RoboDK station: kr30 cnc 072119 adjusting.rdk

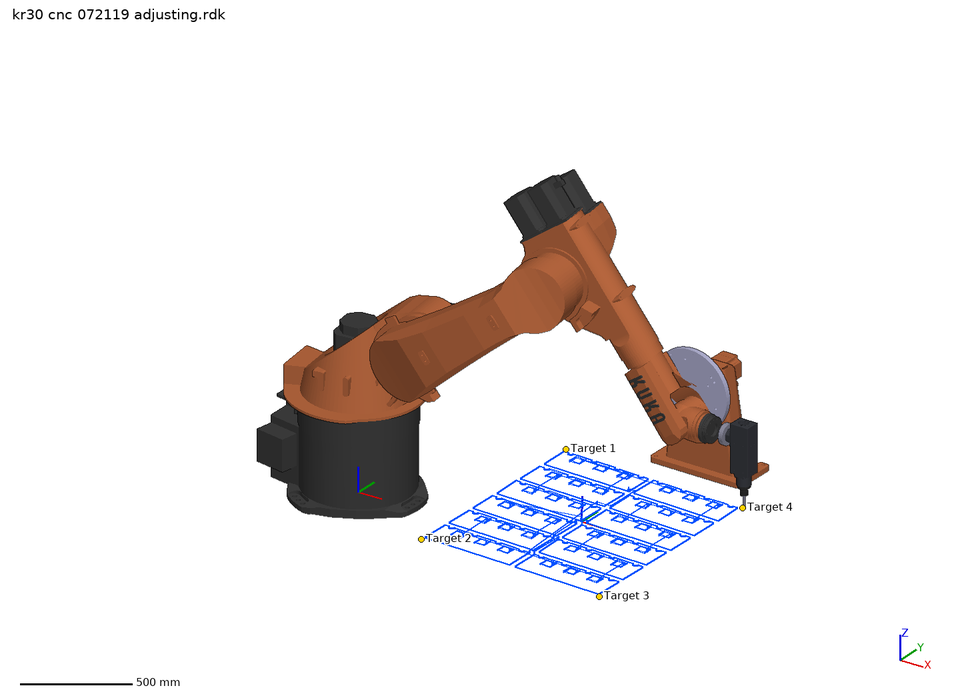
[picture v0: the station drawn from its stored meshes, robots at their saved joint values, targets as dots, program paths as lines]
Station kr30 cnc 072119 adjusting. Poses are relative to the parent item; angles as X-Y-Z fixed-axis rotations.
  - frame GIGASHEEN 7th Axis Base at (0, 0, 0) mm
    - robot KUKA KP1 MD250: 1 axes, payload 250 kg
        modified DH rows (alpha deg, a mm, theta deg, d mm): 0, 0, 0, 0
        base shift (1587.22, 296.05, 828) mm, rotated rx 0 ry 90 rz -90 deg
        joint limits [-3600] to [3600]; home [0]; saved at [1119.52]
      - frame Turntable Base at (243.9, -362.78, 658.66) mm, rotated rx -90.25 ry 0 rz 49.48 deg
  - frame GIGASHEEN Base at (0, 0, 0) mm
    - robot GIGASHEEN (model KUKA KR 30 HA): 6 axes, payload 30 kg, reach 2033 mm, repeatability 0.05 mm, weight 665 kg
        modified DH rows (alpha deg, a mm, theta deg, d mm): 0, 0, 0, 815; -90, 350, 0, 0; 0, 850, -90, 0; -90, 145, 0, 820; 90, 0, 0, 0; -90, 0, 180, 170
        joint limits [-185, -135, -120, -350, -119, -350] to [185, 35, 158, 350, 119, 350]; home [0, -90, 90, 0, 0, 0]; saved at [-6.898, -35.989, 90.741, -8.88, -55.221, 5.167]
      - tool 1/2" End Mill TCP, TCP at (337.71, -2.2, 160.57) mm, rotated rx 0 ry 90 rz 0 deg, size 415.8 x 102 x 153.6 mm
    - target Target 1 (joint target) at (982.46, 202.21, 406.25) mm, rotated rx -179.95 ry 0.15 rz -89.48 deg; joints [7.49, -59.642, 144.935, 97.969, -90.801, -4.608] of GIGASHEEN
    - target Target 2 (joint target) at (986.83, -921.64, 412.07) mm, rotated rx -179.94 ry 0.15 rz -89.48 deg; joints [51.766, -38.608, 94.384, 136.851, -116.554, -22.567] of GIGASHEEN
    - target Target 3 (joint target) at (1949.02, -919.97, 396.91) mm, rotated rx -179.94 ry 0.14 rz 179.61 deg; joints [29.5, -22.76, 62.288, 41.088, -47.759, -30.404] of GIGASHEEN
    - target Target 4 (joint target) at (1949.02, 190.94, 391.63) mm, rotated rx -179.94 ry 0.14 rz 179.61 deg; joints [-6.898, -35.989, 90.741, -8.88, -55.221, 5.167] of GIGASHEEN
  - machining project Machining Settings: C:/Users/liqui/OneDrive/Desktop/first half pipe jig.apt | rotZ(0) | rotX(0)*rotY(0) | rotZ(0)
  - program Machining (1954 instructions, listed below)
  - program Prog2 (4 instructions, listed below)
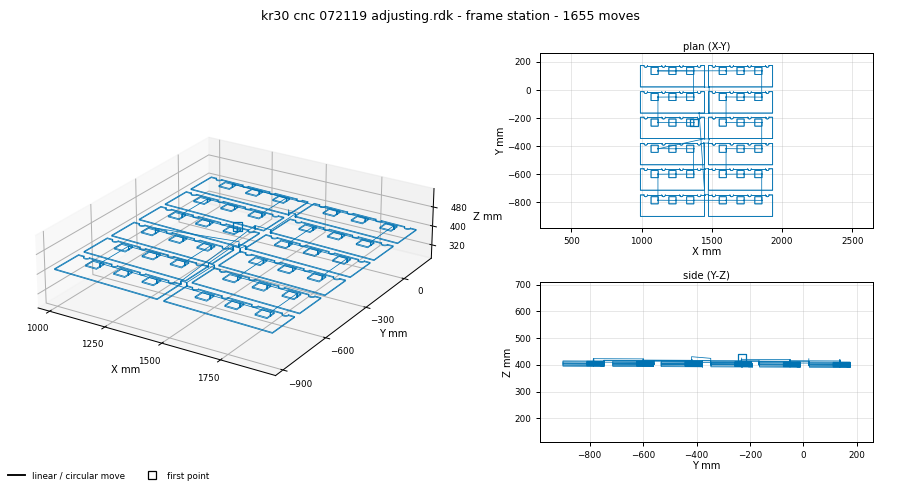
[picture p0: tool path of kr30 cnc 072119 adjusting.rdk in frame station, 1655 of 1659 moves have a stored position in this frame; points joined in program order, loops and branches not executed]

--- program Machining (robot GIGASHEEN) ---
  Smooth(0)
  Set Ref.: Turntable Base
  Set Tool: 1/2" End Mill TCP
  Show 1/2" End Mill TCP
  Print: /'1001'
  Print: /''
  Print: /'2D Contour2'
  Set speed (500.0 mm/s)
  MoveJ 1 to (-92.16, 131.49, 15) mm, rotated rx -180 ry 0 rz -179 deg; joints [17.436, -76.67, 121.961, 23.843, -47.841, -16.522]
  MoveL 2 to (-92.16, 131.49, 15) mm, rotated rx -180 ry 0 rz -179 deg; joints [17.436, -76.67, 121.961, 23.843, -47.841, -16.522]
  MoveL 3 to (-92.16, 131.49, 15) mm, rotated rx -180 ry 0 rz -179 deg; joints [17.436, -76.67, 121.961, 23.843, -47.841, -16.522]
  Set speed (500.0 mm/s)
  MoveL 4 to (-92.16, 131.49, 6) mm, rotated rx 180 ry 0 rz -179 deg; joints [17.436, -76.289, 122.229, 23.608, -48.436, -16.171]
  Set speed (25.4 mm/s)
  MoveL 5 to (-92.16, 131.49, -3.54) mm, rotated rx 180 ry 0 rz -179 deg; joints [17.436, -75.878, 122.507, 23.368, -49.068, -15.806]
  MoveC 6 to (-91.98, 131.48, -3.99) mm, rotated rx -180 ry 0 rz -179 deg; joints [17.434, -75.848, 122.506, 23.355, -49.094, -15.788] to (-91.53, 131.49, -4.17) mm, rotated rx -180 ry 0 rz -179 deg; joints [17.428, -75.815, 122.478, 23.345, -49.097, -15.78]
  Set speed (50.8 mm/s)
  MoveL 7 to (-90.89, 131.49, -4.18) mm, rotated rx -180 ry 0 rz -179 deg; joints [17.42, -75.779, 122.432, 23.338, -49.085, -15.779]
  MoveC 8 to (-90.44, 131.3, -4.18) mm, rotated rx -180 ry 0 rz -179 deg; joints [17.422, -75.751, 122.395, 23.344, -49.077, -15.786] to (-90.26, 130.85, -4.17) mm, rotated rx -180 ry 0 rz -179 deg; joints [17.44, -75.733, 122.371, 23.369, -49.077, -15.803]
  MoveL 9 to (-90.26, 105.45, -4.18) mm, rotated rx 180 ry 0 rz -179 deg; joints [18.57, -75.299, 121.799, 24.851, -49.269, -16.815]
  MoveL 10 to (-141.06, 105.45, -4.17) mm, rotated rx -180 ry 0 rz -179 deg; joints [19.31, -78.143, 125.477, 25.479, -50.238, -16.95]
  MoveL 11 to (-141.06, 156.25, -4.17) mm, rotated rx -180 ry 0 rz -179 deg; joints [16.952, -79.034, 126.595, 22.442, -49.797, -14.928]
  MoveL 12 to (-90.26, 156.25, -4.17) mm, rotated rx -180 ry 0 rz -179 deg; joints [16.296, -76.14, 122.904, 21.865, -48.892, -14.78]
  MoveL 13 to (-90.26, 130.85, -4.17) mm, rotated rx -180 ry 0 rz -179 deg; joints [17.44, -75.733, 122.371, 23.369, -49.077, -15.803]
  MoveC 14 to (-90.44, 130.4, -4.17) mm, rotated rx -180 ry 0 rz -179 deg; joints [17.462, -75.736, 122.375, 23.397, -49.084, -15.822] to (-90.89, 130.21, -4.18) mm, rotated rx -180 ry 0 rz -179 deg; joints [17.477, -75.758, 122.404, 23.413, -49.094, -15.83]
  MoveL 15 to (-91.53, 130.21, -4.18) mm, rotated rx 180 ry 0 rz -179 deg; joints [17.485, -75.794, 122.451, 23.42, -49.107, -15.831]
  MoveC 16 to (-91.98, 130.22, -3.99) mm, rotated rx -180 ry 0 rz -179 deg; joints [17.491, -75.827, 122.479, 23.429, -49.103, -15.839] to (-92.16, 130.22, -3.54) mm, rotated rx -180 ry 0 rz -179 deg; joints [17.493, -75.857, 122.479, 23.442, -49.077, -15.857]
  Set speed (500.0 mm/s)
  MoveL 17 to (-92.16, 130.22, 5) mm, rotated rx -180 ry 0 rz -179 deg; joints [17.493, -76.225, 122.231, 23.658, -48.512, -16.184]
  MoveL 18 to (-92.16, 131.49, 5) mm, rotated rx 180 ry 0 rz -179 deg; joints [17.436, -76.246, 122.259, 23.583, -48.502, -16.132]
  Set speed (25.4 mm/s)
  MoveL 19 to (-92.16, 131.49, 1.82) mm, rotated rx -180 ry 0 rz -179 deg; joints [17.436, -76.11, 122.352, 23.502, -48.712, -16.01]
  MoveL 20 to (-92.16, 131.49, -7.72) mm, rotated rx -180 ry 0 rz -179 deg; joints [17.436, -75.696, 122.626, 23.265, -49.345, -15.648]
  MoveC 21 to (-91.98, 131.49, -8.16) mm, rotated rx 180 ry 0 rz -179 deg; joints [17.434, -75.666, 122.625, 23.252, -49.371, -15.631] to (-91.53, 131.49, -8.35) mm, rotated rx -180 ry 0 rz -179 deg; joints [17.428, -75.632, 122.597, 23.242, -49.374, -15.623]
  Set speed (50.8 mm/s)
  MoveL 22 to (-90.89, 131.49, -8.35) mm, rotated rx -180 ry 0 rz -179 deg; joints [17.42, -75.597, 122.551, 23.235, -49.362, -15.622]
  MoveC 23 to (-90.44, 131.3, -8.35) mm, rotated rx -180 ry 0 rz -179 deg; joints [17.422, -75.569, 122.513, 23.242, -49.354, -15.629] to (-90.26, 130.85, -8.35) mm, rotated rx 180 ry 0 rz -179 deg; joints [17.44, -75.551, 122.49, 23.266, -49.354, -15.646]
  MoveL 24 to (-90.26, 105.45, -8.35) mm, rotated rx -180 ry 0 rz -179 deg; joints [18.57, -75.118, 121.917, 24.743, -49.54, -16.65]
  MoveL 25 to (-141.06, 105.45, -8.35) mm, rotated rx -180 ry 0 rz -179 deg; joints [19.31, -77.953, 125.598, 25.368, -50.519, -16.777]
  MoveL 26 to (-141.06, 156.25, -8.35) mm, rotated rx -180 ry 0 rz -179 deg; joints [16.952, -78.842, 126.718, 22.341, -50.089, -14.771]
  MoveL 27 to (-90.26, 156.25, -8.35) mm, rotated rx 180 ry 0 rz -179 deg; joints [16.296, -75.956, 123.023, 21.767, -49.173, -14.631]
  MoveL 28 to (-90.26, 130.85, -8.35) mm, rotated rx 180 ry 0 rz -179 deg; joints [17.44, -75.551, 122.49, 23.266, -49.354, -15.646]
  MoveC 29 to (-90.44, 130.4, -8.35) mm, rotated rx -180 ry 0 rz -179 deg; joints [17.462, -75.554, 122.494, 23.294, -49.36, -15.664] to (-90.89, 130.21, -8.35) mm, rotated rx -180 ry 0 rz -179 deg; joints [17.477, -75.576, 122.523, 23.31, -49.371, -15.672]
  MoveL 30 to (-91.53, 130.21, -8.35) mm, rotated rx -180 ry 0 rz -179 deg; joints [17.485, -75.611, 122.57, 23.317, -49.383, -15.673]
  MoveC 31 to (-91.98, 130.22, -8.16) mm, rotated rx 180 ry 0 rz -179 deg; joints [17.491, -75.645, 122.598, 23.326, -49.38, -15.681] to (-92.16, 130.22, -7.72) mm, rotated rx -180 ry 0 rz -179 deg; joints [17.493, -75.675, 122.598, 23.339, -49.354, -15.698]
  Set speed (500.0 mm/s)
  MoveL 32 to (-92.16, 130.22, 6) mm, rotated rx 180 ry 0 rz -179 deg; joints [17.493, -76.268, 122.202, 23.684, -48.446, -16.223]
  MoveL 33 to (-219.16, 131.49, 6) mm, rotated rx -180 ry 0 rz -179 deg; joints [19.301, -83.624, 131.192, 25.384, -50.447, -16.812]
  Set speed (25.4 mm/s)
  MoveL 34 to (-219.16, 131.49, -3.54) mm, rotated rx -180 ry 0 rz -179 deg; joints [19.301, -83.162, 131.493, 25.118, -51.137, -16.392]
  MoveC 35 to (-218.98, 131.49, -3.99) mm, rotated rx -180 ry 0 rz -179 deg; joints [19.298, -83.129, 131.494, 25.103, -51.167, -16.371] to (-218.53, 131.48, -4.17) mm, rotated rx -180 ry 0 rz -179 deg; joints [19.29, -83.093, 131.469, 25.09, -51.175, -16.359]
  Set speed (50.8 mm/s)
  MoveL 36 to (-217.89, 131.49, -4.18) mm, rotated rx -180 ry 0 rz -179 deg; joints [19.28, -83.056, 131.426, 25.079, -51.167, -16.355]
  MoveC 37 to (-217.44, 131.3, -4.17) mm, rotated rx -180 ry 0 rz -179 deg; joints [19.282, -83.026, 131.392, 25.083, -51.163, -16.359] to (-217.26, 130.85, -4.17) mm, rotated rx -180 ry 0 rz -179 deg; joints [19.301, -83.006, 131.369, 25.108, -51.166, -16.375]
  MoveL 38 to (-217.26, 105.45, -4.17) mm, rotated rx -180 ry 0 rz -179 deg; joints [20.54, -82.498, 130.777, 26.656, -51.45, -17.372]
  MoveL 39 to (-268.06, 105.45, -4.18) mm, rotated rx 180 ry 0 rz -179 deg; joints [21.453, -85.484, 134.171, 27.617, -52.089, -17.82]
  MoveL 40 to (-268.06, 156.25, -4.18) mm, rotated rx 180 ry 0 rz -179 deg; joints [18.856, -86.551, 135.335, 24.418, -51.424, -15.806]
  MoveL 41 to (-217.26, 156.25, -4.18) mm, rotated rx -180 ry 0 rz -179 deg; joints [18.043, -83.485, 131.921, 23.527, -50.889, -15.358]
  MoveL 42 to (-217.26, 130.85, -4.17) mm, rotated rx -180 ry 0 rz -179 deg; joints [19.301, -83.006, 131.369, 25.108, -51.166, -16.375]
  MoveC 43 to (-217.44, 130.4, -4.18) mm, rotated rx 180 ry 0 rz -179 deg; joints [19.326, -83.008, 131.371, 25.138, -51.173, -16.394] to (-217.89, 130.22, -4.17) mm, rotated rx -180 ry 0 rz -179 deg; joints [19.342, -83.031, 131.398, 25.157, -51.181, -16.405]
  MoveL 44 to (-218.53, 130.22, -4.18) mm, rotated rx 180 ry 0 rz -179 deg; joints [19.353, -83.068, 131.441, 25.168, -51.189, -16.41]
  MoveC 45 to (-218.98, 130.21, -3.99) mm, rotated rx -180 ry 0 rz -179 deg; joints [19.36, -83.104, 131.466, 25.181, -51.182, -16.421] to (-219.16, 130.21, -3.54) mm, rotated rx -180 ry 0 rz -179 deg; joints [19.363, -83.137, 131.464, 25.196, -51.151, -16.442]
  Set speed (500.0 mm/s)
  MoveL 46 to (-219.16, 130.22, 5) mm, rotated rx 180 ry 0 rz -179 deg; joints [19.363, -83.551, 131.196, 25.434, -50.534, -16.819]
  MoveL 47 to (-219.16, 131.48, 5) mm, rotated rx -180 ry 0 rz -179 deg; joints [19.301, -83.576, 131.224, 25.355, -50.519, -16.768]
  Set speed (25.4 mm/s)
  MoveL 48 to (-219.16, 131.48, 1.82) mm, rotated rx -180 ry 0 rz -179 deg; joints [19.301, -83.423, 131.325, 25.266, -50.749, -16.627]
  MoveL 49 to (-219.16, 131.49, -7.72) mm, rotated rx -180 ry 0 rz -179 deg; joints [19.301, -82.956, 131.622, 25.004, -51.44, -16.21]
  MoveC 50 to (-218.98, 131.49, -8.16) mm, rotated rx -180 ry 0 rz -179 deg; joints [19.298, -82.923, 131.623, 24.989, -51.47, -16.189] to (-218.53, 131.49, -8.35) mm, rotated rx -180 ry 0 rz -179 deg; joints [19.29, -82.888, 131.598, 24.977, -51.478, -16.178]
  Set speed (50.8 mm/s)
  MoveL 51 to (-217.89, 131.48, -8.35) mm, rotated rx -180 ry 0 rz -179 deg; joints [19.28, -82.85, 131.555, 24.966, -51.47, -16.174]
  MoveC 52 to (-217.44, 131.3, -8.35) mm, rotated rx -180 ry 0 rz -179 deg; joints [19.282, -82.82, 131.52, 24.97, -51.466, -16.178] to (-217.26, 130.85, -8.35) mm, rotated rx -180 ry 0 rz -179 deg; joints [19.301, -82.801, 131.497, 24.994, -51.468, -16.194]
  MoveL 53 to (-217.26, 105.45, -8.35) mm, rotated rx -180 ry 0 rz -179 deg; joints [20.54, -82.294, 130.905, 26.539, -51.747, -17.182]
  MoveL 54 to (-268.06, 105.45, -8.35) mm, rotated rx -180 ry 0 rz -179 deg; joints [21.453, -85.271, 134.303, 27.493, -52.396, -17.618]
  MoveL 55 to (-268.06, 156.25, -8.35) mm, rotated rx -180 ry 0 rz -179 deg; joints [18.856, -86.334, 135.469, 24.303, -51.745, -15.621]
  MoveL 56 to (-217.26, 156.25, -8.35) mm, rotated rx -180 ry 0 rz -179 deg; joints [18.043, -83.278, 132.05, 23.419, -51.197, -15.185]
  MoveL 57 to (-217.26, 130.85, -8.35) mm, rotated rx -180 ry 0 rz -179 deg; joints [19.301, -82.801, 131.497, 24.994, -51.468, -16.194]
  MoveC 58 to (-217.44, 130.4, -8.35) mm, rotated rx -180 ry 0 rz -179 deg; joints [19.326, -82.803, 131.5, 25.025, -51.476, -16.213] to (-217.89, 130.22, -8.35) mm, rotated rx 180 ry 0 rz -179 deg; joints [19.342, -82.826, 131.526, 25.044, -51.484, -16.223]
  MoveL 59 to (-218.53, 130.21, -8.35) mm, rotated rx -180 ry 0 rz -179 deg; joints [19.353, -82.863, 131.57, 25.055, -51.492, -16.228]
  MoveC 60 to (-218.98, 130.21, -8.16) mm, rotated rx -180 ry 0 rz -179 deg; joints [19.36, -82.898, 131.595, 25.067, -51.484, -16.239] to (-219.16, 130.22, -7.72) mm, rotated rx 180 ry 0 rz -179 deg; joints [19.363, -82.932, 131.593, 25.082, -51.454, -16.26]
  Set speed (500.0 mm/s)
  MoveL 61 to (-219.16, 130.21, 6) mm, rotated rx -180 ry 0 rz -179 deg; joints [19.363, -83.599, 131.164, 25.462, -50.462, -16.863]
  MoveL 62 to (-346.16, 131.48, 6) mm, rotated rx -180 ry 0 rz -179 deg; joints [21.621, -91.451, 139.452, 28.072, -51.536, -18.353]
  Set speed (25.4 mm/s)
  MoveL 63 to (-346.16, 131.48, -3.54) mm, rotated rx -180 ry 0 rz -179 deg; joints [21.621, -90.932, 139.786, 27.76, -52.288, -17.847]
  MoveC 64 to (-345.98, 131.49, -3.99) mm, rotated rx 180 ry 0 rz -179 deg; joints [21.617, -90.896, 139.79, 27.741, -52.323, -17.82] to (-345.53, 131.48, -4.17) mm, rotated rx -180 ry 0 rz -179 deg; joints [21.608, -90.857, 139.768, 27.724, -52.335, -17.803]
  Set speed (50.8 mm/s)
  MoveL 65 to (-344.89, 131.49, -4.18) mm, rotated rx -180 ry 0 rz -179 deg; joints [21.595, -90.816, 139.728, 27.708, -52.332, -17.793]
  MoveC 66 to (-344.44, 131.3, -4.17) mm, rotated rx 180 ry 0 rz -179 deg; joints [21.596, -90.783, 139.696, 27.709, -52.333, -17.793] to (-344.26, 130.85, -4.18) mm, rotated rx 180 ry 0 rz -179 deg; joints [21.617, -90.76, 139.673, 27.733, -52.339, -17.808]
  MoveL 67 to (-344.26, 105.45, -4.17) mm, rotated rx -180 ry 0 rz -179 deg; joints [22.984, -90.134, 139.054, 29.366, -52.775, -18.799]
  MoveL 68 to (-395.06, 105.45, -4.18) mm, rotated rx -180 ry 0 rz -179 deg; joints [24.132, -93.379, 142.168, 30.774, -53.04, -19.7]
  MoveL 69 to (-395.06, 156.25, -4.18) mm, rotated rx -180 ry 0 rz -179 deg; joints [21.254, -94.725, 143.389, 27.385, -52.009, -17.686]
  MoveL 70 to (-344.26, 156.25, -4.18) mm, rotated rx -180 ry 0 rz -179 deg; joints [20.224, -91.353, 140.251, 26.054, -51.913, -16.782]
  MoveL 71 to (-344.26, 130.85, -4.18) mm, rotated rx 180 ry 0 rz -179 deg; joints [21.617, -90.76, 139.673, 27.733, -52.339, -17.808]
  MoveC 72 to (-344.44, 130.4, -4.18) mm, rotated rx -180 ry 0 rz -179 deg; joints [21.645, -90.761, 139.674, 27.767, -52.348, -17.829] to (-344.89, 130.22, -4.18) mm, rotated rx -180 ry 0 rz -179 deg; joints [21.664, -90.786, 139.698, 27.79, -52.354, -17.843]
  MoveL 73 to (-345.53, 130.22, -4.18) mm, rotated rx 180 ry 0 rz -179 deg; joints [21.677, -90.826, 139.738, 27.806, -52.357, -17.853]
  MoveC 74 to (-345.98, 130.21, -3.99) mm, rotated rx 180 ry 0 rz -179 deg; joints [21.686, -90.865, 139.76, 27.824, -52.344, -17.87] to (-346.16, 130.22, -3.54) mm, rotated rx -180 ry 0 rz -179 deg; joints [21.69, -90.902, 139.756, 27.843, -52.31, -17.897]
  Set speed (500.0 mm/s)
  MoveL 75 to (-346.16, 130.22, 5) mm, rotated rx -180 ry 0 rz -179 deg; joints [21.69, -91.366, 139.458, 28.123, -51.637, -18.351]
  MoveL 76 to (-346.16, 131.48, 5) mm, rotated rx -180 ry 0 rz -179 deg; joints [21.621, -91.397, 139.488, 28.039, -51.614, -18.3]
  Set speed (25.4 mm/s)
  MoveL 77 to (-346.16, 131.49, 1.83) mm, rotated rx -180 ry 0 rz -179 deg; joints [21.621, -91.225, 139.599, 27.934, -51.864, -18.13]
  MoveL 78 to (-346.16, 131.49, -7.72) mm, rotated rx 180 ry 0 rz -179 deg; joints [21.621, -90.702, 139.929, 27.626, -52.619, -17.627]
  MoveC 79 to (-345.98, 131.49, -8.16) mm, rotated rx 180 ry 0 rz -179 deg; joints [21.617, -90.665, 139.933, 27.607, -52.654, -17.601] to (-345.53, 131.49, -8.35) mm, rotated rx 180 ry 0 rz -179 deg; joints [21.608, -90.626, 139.911, 27.59, -52.666, -17.584]
  Set speed (50.8 mm/s)
  MoveL 80 to (-344.89, 131.48, -8.35) mm, rotated rx -180 ry 0 rz -179 deg; joints [21.595, -90.585, 139.871, 27.575, -52.663, -17.575]
  MoveC 81 to (-344.44, 131.3, -8.35) mm, rotated rx -180 ry 0 rz -179 deg; joints [21.596, -90.552, 139.838, 27.576, -52.664, -17.575] to (-344.26, 130.85, -8.35) mm, rotated rx 180 ry 0 rz -179 deg; joints [21.617, -90.53, 139.816, 27.6, -52.67, -17.59]
  MoveL 82 to (-344.26, 105.45, -8.35) mm, rotated rx -180 ry 0 rz -179 deg; joints [22.984, -89.906, 139.195, 29.229, -53.097, -18.572]
  MoveL 83 to (-395.06, 105.45, -8.35) mm, rotated rx 180 ry 0 rz -179 deg; joints [24.132, -93.14, 142.316, 30.626, -53.373, -19.453]
  MoveL 84 to (-395.06, 156.25, -8.35) mm, rotated rx -180 ry 0 rz -179 deg; joints [21.254, -94.482, 143.541, 27.245, -52.359, -17.457]
  MoveL 85 to (-344.26, 156.25, -8.35) mm, rotated rx -180 ry 0 rz -179 deg; joints [20.224, -91.12, 140.395, 25.925, -52.251, -16.573]
  MoveL 86 to (-344.26, 130.85, -8.35) mm, rotated rx 180 ry 0 rz -179 deg; joints [21.617, -90.53, 139.816, 27.6, -52.67, -17.59]
  MoveC 87 to (-344.44, 130.4, -8.35) mm, rotated rx -180 ry 0 rz -179 deg; joints [21.645, -90.531, 139.817, 27.634, -52.679, -17.61] to (-344.89, 130.21, -8.35) mm, rotated rx 180 ry 0 rz -179 deg; joints [21.664, -90.555, 139.841, 27.657, -52.684, -17.624]
  MoveL 88 to (-345.53, 130.22, -8.35) mm, rotated rx -180 ry 0 rz -179 deg; joints [21.677, -90.595, 139.881, 27.673, -52.688, -17.634]
  MoveC 89 to (-345.98, 130.22, -8.16) mm, rotated rx 180 ry 0 rz -179 deg; joints [21.686, -90.634, 139.903, 27.69, -52.675, -17.651] to (-346.16, 130.21, -7.72) mm, rotated rx -180 ry 0 rz -179 deg; joints [21.69, -90.671, 139.899, 27.709, -52.641, -17.677]
  Set speed (500.0 mm/s)
  MoveL 90 to (-346.16, 130.22, 6) mm, rotated rx 180 ry 0 rz -179 deg; joints [21.69, -91.42, 139.423, 28.156, -51.558, -18.405]
  MoveL 91 to (-346.16, 313.35, 6) mm, rotated rx -180 ry 0 rz -179 deg; joints [11.148, -94.869, 142.627, 14.906, -48.733, -9.958]
  Set speed (25.4 mm/s)
  MoveL 92 to (-346.16, 313.36, -3.54) mm, rotated rx 180 ry 0 rz -179 deg; joints [11.148, -94.327, 142.977, 14.709, -49.594, -9.657]
  MoveC 93 to (-345.98, 313.36, -3.99) mm, rotated rx 180 ry 0 rz -179 deg; joints [11.146, -94.288, 142.981, 14.697, -49.636, -9.641] to (-345.53, 313.35, -4.17) mm, rotated rx -180 ry 0 rz -179 deg; joints [11.142, -94.246, 142.959, 14.687, -49.655, -9.63]
  Set speed (50.8 mm/s)
  MoveL 94 to (-344.89, 313.36, -4.18) mm, rotated rx 180 ry 0 rz -179 deg; joints [11.135, -94.201, 142.919, 14.677, -49.658, -9.623]
  MoveC 95 to (-344.44, 313.17, -4.18) mm, rotated rx -180 ry 0 rz -179 deg; joints [11.141, -94.167, 142.888, 14.684, -49.662, -9.627] to (-344.26, 312.72, -4.18) mm, rotated rx -180 ry 0 rz -179 deg; joints [11.166, -94.148, 142.871, 14.716, -49.668, -9.648]
  MoveL 96 to (-344.26, 287.32, -4.18) mm, rotated rx 180 ry 0 rz -179 deg; joints [12.685, -93.803, 142.558, 16.665, -49.969, -10.899]
  MoveL 97 to (-395.06, 287.32, -4.18) mm, rotated rx -180 ry 0 rz -179 deg; joints [13.345, -97.456, 145.743, 17.629, -49.652, -11.626]
  MoveL 98 to (-395.06, 338.12, -4.18) mm, rotated rx -180 ry 0 rz -179 deg; joints [10.127, -98.178, 146.337, 13.482, -48.954, -8.947]
  MoveL 99 to (-344.26, 338.12, -4.17) mm, rotated rx -180 ry 0 rz -179 deg; joints [9.633, -94.446, 143.14, 12.732, -49.4, -8.365]
  MoveL 100 to (-344.26, 312.72, -4.17) mm, rotated rx -180 ry 0 rz -179 deg; joints [11.166, -94.148, 142.871, 14.716, -49.668, -9.648]
  MoveC 101 to (-344.44, 312.27, -4.18) mm, rotated rx -180 ry 0 rz -179 deg; joints [11.195, -94.155, 142.878, 14.754, -49.672, -9.672] to (-344.89, 312.09, -4.18) mm, rotated rx 180 ry 0 rz -179 deg; joints [11.211, -94.185, 142.904, 14.775, -49.672, -9.686]
  MoveL 102 to (-345.53, 312.09, -4.18) mm, rotated rx -180 ry 0 rz -179 deg; joints [11.218, -94.23, 142.945, 14.785, -49.669, -9.694]
  MoveC 103 to (-345.98, 312.09, -3.99) mm, rotated rx -180 ry 0 rz -179 deg; joints [11.223, -94.272, 142.967, 14.796, -49.65, -9.705] to (-346.16, 312.08, -3.54) mm, rotated rx -180 ry 0 rz -179 deg; joints [11.225, -94.311, 142.962, 14.808, -49.609, -9.721]
  Set speed (500.0 mm/s)
  MoveL 104 to (-346.16, 312.09, 5) mm, rotated rx 180 ry 0 rz -179 deg; joints [11.225, -94.796, 142.65, 14.985, -48.838, -9.992]
  MoveL 105 to (-346.16, 313.36, 5) mm, rotated rx 180 ry 0 rz -179 deg; joints [11.148, -94.813, 142.664, 14.885, -48.823, -9.926]
  Set speed (25.4 mm/s)
  MoveL 106 to (-346.16, 313.36, 1.82) mm, rotated rx -180 ry 0 rz -179 deg; joints [11.148, -94.633, 142.781, 14.819, -49.109, -9.826]
  MoveL 107 to (-346.16, 313.35, -7.71) mm, rotated rx -180 ry 0 rz -179 deg; joints [11.148, -94.086, 143.128, 14.625, -49.974, -9.527]
  MoveC 108 to (-345.98, 313.36, -8.16) mm, rotated rx -180 ry 0 rz -179 deg; joints [11.146, -94.047, 143.132, 14.614, -50.015, -9.511] to (-345.53, 313.36, -8.35) mm, rotated rx -180 ry 0 rz -179 deg; joints [11.142, -94.004, 143.11, 14.603, -50.034, -9.501]
  Set speed (50.8 mm/s)
  MoveL 109 to (-344.89, 313.35, -8.35) mm, rotated rx -180 ry 0 rz -179 deg; joints [11.135, -93.959, 143.069, 14.593, -50.037, -9.494]
  MoveC 110 to (-344.44, 313.17, -8.35) mm, rotated rx -180 ry 0 rz -179 deg; joints [11.141, -93.925, 143.038, 14.601, -50.041, -9.498] to (-344.26, 312.72, -8.35) mm, rotated rx -180 ry 0 rz -179 deg; joints [11.166, -93.907, 143.021, 14.633, -50.047, -9.518]
  MoveL 111 to (-344.26, 287.32, -8.35) mm, rotated rx -180 ry 0 rz -179 deg; joints [12.685, -93.563, 142.707, 16.572, -50.342, -10.754]
  MoveL 112 to (-395.06, 287.32, -8.35) mm, rotated rx -180 ry 0 rz -179 deg; joints [13.345, -97.205, 145.9, 17.525, -50.041, -11.464]
  MoveL 113 to (-395.06, 338.12, -8.35) mm, rotated rx 180 ry 0 rz -179 deg; joints [10.127, -97.925, 146.497, 13.399, -49.355, -8.82]
  MoveL 114 to (-344.26, 338.12, -8.35) mm, rotated rx -180 ry 0 rz -179 deg; joints [9.633, -94.204, 143.291, 12.658, -49.783, -8.251]
  MoveL 115 to (-344.26, 312.72, -8.35) mm, rotated rx -180 ry 0 rz -179 deg; joints [11.166, -93.907, 143.021, 14.633, -50.047, -9.518]
  MoveC 116 to (-344.44, 312.27, -8.35) mm, rotated rx -180 ry 0 rz -179 deg; joints [11.195, -93.914, 143.028, 14.67, -50.051, -9.542] to (-344.89, 312.08, -8.35) mm, rotated rx -180 ry 0 rz -179 deg; joints [11.211, -93.943, 143.054, 14.691, -50.051, -9.556]
  MoveL 117 to (-345.53, 312.08, -8.35) mm, rotated rx -180 ry 0 rz -179 deg; joints [11.218, -93.988, 143.095, 14.701, -50.048, -9.563]
  MoveC 118 to (-345.98, 312.08, -8.16) mm, rotated rx -180 ry 0 rz -179 deg; joints [11.223, -94.031, 143.117, 14.712, -50.029, -9.574] to (-346.16, 312.08, -7.72) mm, rotated rx -180 ry 0 rz -179 deg; joints [11.225, -94.07, 143.113, 14.724, -49.988, -9.59]
  Set speed (500.0 mm/s)
  MoveL 119 to (-346.16, 312.08, 6) mm, rotated rx -180 ry 0 rz -179 deg; joints [11.225, -94.852, 142.613, 15.006, -48.748, -10.024]
  MoveL 120 to (-219.16, 313.36, 6) mm, rotated rx -180 ry 0 rz -179 deg; joints [9.941, -86.348, 134.223, 13.295, -48.648, -8.873]
  Set speed (25.4 mm/s)
  MoveL 121 to (-219.16, 313.36, -3.54) mm, rotated rx -180 ry 0 rz -179 deg; joints [9.941, -85.865, 134.534, 13.138, -49.421, -8.633]
  MoveC 122 to (-218.98, 313.36, -3.99) mm, rotated rx 180 ry 0 rz -179 deg; joints [9.939, -85.831, 134.535, 13.129, -49.456, -8.621] to (-218.53, 313.36, -4.17) mm, rotated rx -180 ry 0 rz -179 deg; joints [9.935, -85.793, 134.51, 13.121, -49.468, -8.614]
  Set speed (50.8 mm/s)
  MoveL 123 to (-217.89, 313.36, -4.17) mm, rotated rx -180 ry 0 rz -179 deg; joints [9.93, -85.753, 134.466, 13.115, -49.463, -8.611]
  MoveC 124 to (-217.44, 313.17, -4.18) mm, rotated rx 180 ry 0 rz -179 deg; joints [9.936, -85.723, 134.433, 13.124, -49.461, -8.617] to (-217.26, 312.72, -4.18) mm, rotated rx 180 ry 0 rz -179 deg; joints [9.959, -85.707, 134.416, 13.153, -49.463, -8.636]
  MoveL 125 to (-217.26, 287.32, -4.17) mm, rotated rx -180 ry 0 rz -179 deg; joints [11.305, -85.436, 134.118, 14.905, -49.652, -9.777]
  MoveL 126 to (-268.06, 287.32, -4.18) mm, rotated rx 180 ry 0 rz -179 deg; joints [11.816, -88.674, 137.573, 15.516, -49.95, -10.128]
  MoveL 127 to (-268.06, 338.12, -4.18) mm, rotated rx 180 ry 0 rz -179 deg; joints [8.984, -89.225, 138.138, 11.846, -49.523, -7.754]
  MoveL 128 to (-217.26, 338.12, -4.18) mm, rotated rx -180 ry 0 rz -179 deg; joints [8.602, -85.94, 134.672, 11.38, -49.294, -7.478]
  MoveL 129 to (-217.26, 312.72, -4.18) mm, rotated rx 180 ry 0 rz -179 deg; joints [9.959, -85.707, 134.416, 13.153, -49.463, -8.636]
  MoveC 130 to (-217.44, 312.27, -4.17) mm, rotated rx -180 ry 0 rz -179 deg; joints [9.984, -85.714, 134.424, 13.186, -49.467, -8.657] to (-217.89, 312.08, -4.17) mm, rotated rx -180 ry 0 rz -179 deg; joints [9.998, -85.74, 134.453, 13.203, -49.472, -8.668]
  MoveL 131 to (-218.53, 312.08, -4.18) mm, rotated rx -180 ry 0 rz -179 deg; joints [10.003, -85.78, 134.497, 13.209, -49.477, -8.671]
  MoveC 132 to (-218.98, 312.08, -3.99) mm, rotated rx -180 ry 0 rz -179 deg; joints [10.007, -85.818, 134.522, 13.217, -49.465, -8.679] to (-219.16, 312.08, -3.54) mm, rotated rx 180 ry 0 rz -179 deg; joints [10.008, -85.853, 134.52, 13.226, -49.43, -8.691]
  Set speed (500.0 mm/s)
  MoveL 133 to (-219.16, 312.08, 5) mm, rotated rx -180 ry 0 rz -179 deg; joints [10.008, -86.285, 134.242, 13.368, -48.739, -8.907]
  MoveL 134 to (-219.16, 313.35, 5) mm, rotated rx -180 ry 0 rz -179 deg; joints [9.941, -86.298, 134.256, 13.278, -48.729, -8.848]
  Set speed (25.4 mm/s)
  MoveL 135 to (-219.16, 313.36, 1.82) mm, rotated rx -180 ry 0 rz -179 deg; joints [9.941, -86.138, 134.36, 13.226, -48.986, -8.768]
  MoveL 136 to (-219.16, 313.35, -7.72) mm, rotated rx -180 ry 0 rz -179 deg; joints [9.941, -85.651, 134.668, 13.07, -49.759, -8.53]
  MoveC 137 to (-218.98, 313.36, -8.16) mm, rotated rx -180 ry 0 rz -179 deg; joints [9.939, -85.616, 134.669, 13.062, -49.794, -8.517] to (-218.53, 313.36, -8.35) mm, rotated rx -180 ry 0 rz -179 deg; joints [9.935, -85.579, 134.644, 13.054, -49.806, -8.511]
  Set speed (50.8 mm/s)
  MoveL 138 to (-217.89, 313.36, -8.35) mm, rotated rx 180 ry 0 rz -179 deg; joints [9.93, -85.539, 134.6, 13.048, -49.802, -8.507]
  MoveC 139 to (-217.44, 313.17, -8.35) mm, rotated rx 180 ry 0 rz -179 deg; joints [9.936, -85.509, 134.567, 13.057, -49.799, -8.513] to (-217.26, 312.72, -8.35) mm, rotated rx -180 ry 0 rz -179 deg; joints [9.959, -85.493, 134.549, 13.086, -49.801, -8.533]
  MoveL 140 to (-217.26, 287.32, -8.35) mm, rotated rx -180 ry 0 rz -179 deg; joints [11.305, -85.223, 134.251, 14.83, -49.986, -9.661]
  MoveL 141 to (-268.06, 287.32, -8.35) mm, rotated rx 180 ry 0 rz -179 deg; joints [11.816, -88.45, 137.712, 15.435, -50.3, -10.002]
  MoveL 142 to (-268.06, 338.12, -8.35) mm, rotated rx -180 ry 0 rz -179 deg; joints [8.984, -88.999, 138.277, 11.783, -49.88, -7.656]
  MoveL 143 to (-217.26, 338.12, -8.35) mm, rotated rx -180 ry 0 rz -179 deg; joints [8.602, -85.725, 134.805, 11.321, -49.636, -7.388]
  MoveL 144 to (-217.26, 312.72, -8.35) mm, rotated rx -180 ry 0 rz -179 deg; joints [9.959, -85.493, 134.549, 13.086, -49.801, -8.533]
  MoveC 145 to (-217.44, 312.27, -8.35) mm, rotated rx -180 ry 0 rz -179 deg; joints [9.984, -85.5, 134.557, 13.119, -49.806, -8.554] to (-217.89, 312.08, -8.35) mm, rotated rx 180 ry 0 rz -179 deg; joints [9.998, -85.526, 134.586, 13.136, -49.81, -8.564]
  MoveL 146 to (-218.53, 312.09, -8.35) mm, rotated rx -180 ry 0 rz -179 deg; joints [10.003, -85.566, 134.63, 13.142, -49.815, -8.567]
  MoveC 147 to (-218.98, 312.08, -8.16) mm, rotated rx -180 ry 0 rz -179 deg; joints [10.007, -85.604, 134.655, 13.149, -49.803, -8.574] to (-219.16, 312.08, -7.72) mm, rotated rx -180 ry 0 rz -179 deg; joints [10.008, -85.639, 134.654, 13.158, -49.768, -8.587]
  Set speed (500.0 mm/s)
  MoveL 148 to (-219.16, 312.08, 6) mm, rotated rx -180 ry 0 rz -179 deg; joints [10.008, -86.335, 134.209, 13.384, -48.658, -8.932]
  MoveL 149 to (-92.16, 313.35, 6) mm, rotated rx -180 ry 0 rz -179 deg; joints [8.988, -78.58, 125.15, 12.287, -47.233, -8.413]
  Set speed (25.4 mm/s)
  MoveL 150 to (-92.16, 313.36, -3.54) mm, rotated rx 180 ry 0 rz -179 deg; joints [8.988, -78.153, 125.434, 12.15, -47.928, -8.209]
  MoveC 151 to (-91.98, 313.36, -3.99) mm, rotated rx -180 ry 0 rz -179 deg; joints [8.987, -78.121, 125.433, 12.142, -47.957, -8.199] to (-91.53, 313.36, -4.17) mm, rotated rx -180 ry 0 rz -179 deg; joints [8.984, -78.087, 125.405, 12.137, -47.964, -8.194]
  Set speed (50.8 mm/s)
  MoveL 152 to (-90.89, 313.36, -4.18) mm, rotated rx 180 ry 0 rz -179 deg; joints [8.98, -78.049, 125.358, 12.133, -47.953, -8.193]
  MoveC 153 to (-90.44, 313.17, -4.17) mm, rotated rx -180 ry 0 rz -179 deg; joints [8.986, -78.021, 125.323, 12.142, -47.947, -8.201] to (-90.26, 312.72, -4.17) mm, rotated rx -180 ry 0 rz -179 deg; joints [9.006, -78.007, 125.304, 12.17, -47.946, -8.22]
  MoveL 154 to (-90.26, 287.32, -4.17) mm, rotated rx 180 ry 0 rz -179 deg; joints [10.214, -77.781, 125.018, 13.789, -48.071, -9.313]
  MoveL 155 to (-141.06, 287.32, -4.17) mm, rotated rx -180 ry 0 rz -179 deg; joints [10.621, -80.783, 128.739, 14.172, -48.835, -9.437]
  MoveL 156 to (-141.06, 338.12, -4.17) mm, rotated rx -180 ry 0 rz -179 deg; joints [8.094, -81.231, 129.278, 10.825, -48.558, -7.213]
  MoveL 157 to (-90.26, 338.12, -4.17) mm, rotated rx -180 ry 0 rz -179 deg; joints [7.791, -78.201, 125.55, 10.538, -47.834, -7.118]
  MoveL 158 to (-90.26, 312.72, -4.17) mm, rotated rx -180 ry 0 rz -179 deg; joints [9.006, -78.007, 125.304, 12.17, -47.946, -8.22]
  MoveC 159 to (-90.44, 312.27, -4.17) mm, rotated rx -180 ry 0 rz -179 deg; joints [9.028, -78.014, 125.314, 12.2, -47.951, -8.24] to (-90.89, 312.09, -4.17) mm, rotated rx -180 ry 0 rz -179 deg; joints [9.04, -78.039, 125.345, 12.215, -47.959, -8.248]
  MoveL 160 to (-91.53, 312.09, -4.18) mm, rotated rx 180 ry 0 rz -179 deg; joints [9.045, -78.076, 125.392, 12.218, -47.97, -8.249]
  MoveC 161 to (-91.98, 312.09, -3.99) mm, rotated rx 180 ry 0 rz -179 deg; joints [9.048, -78.111, 125.42, 12.224, -47.963, -8.254] to (-92.16, 312.09, -3.54) mm, rotated rx -180 ry 0 rz -179 deg; joints [9.049, -78.142, 125.421, 12.231, -47.934, -8.264]
  Set speed (500.0 mm/s)
  MoveL 162 to (-92.16, 312.09, 5) mm, rotated rx -180 ry 0 rz -179 deg; joints [9.049, -78.525, 125.167, 12.355, -47.312, -8.447]
  MoveL 163 to (-92.16, 313.36, 5) mm, rotated rx 180 ry 0 rz -179 deg; joints [8.988, -78.535, 125.18, 12.273, -47.306, -8.391]
  Set speed (25.4 mm/s)
  MoveL 164 to (-92.16, 313.36, 1.82) mm, rotated rx -180 ry 0 rz -179 deg; joints [8.988, -78.394, 125.275, 12.227, -47.537, -8.323]
  MoveL 165 to (-92.16, 313.36, -7.71) mm, rotated rx 180 ry 0 rz -179 deg; joints [8.988, -77.963, 125.556, 12.091, -48.232, -8.121]
  MoveC 166 to (-91.98, 313.36, -8.16) mm, rotated rx -180 ry 0 rz -179 deg; joints [8.987, -77.932, 125.555, 12.084, -48.262, -8.111] to (-91.53, 313.36, -8.35) mm, rotated rx -180 ry 0 rz -179 deg; joints [8.984, -77.897, 125.527, 12.079, -48.268, -8.107]
  Set speed (50.8 mm/s)
  MoveL 167 to (-90.89, 313.36, -8.35) mm, rotated rx 180 ry 0 rz -179 deg; joints [8.98, -77.86, 125.48, 12.075, -48.258, -8.106]
  MoveC 168 to (-90.44, 313.17, -8.35) mm, rotated rx -180 ry 0 rz -179 deg; joints [8.986, -77.832, 125.445, 12.084, -48.251, -8.113] to (-90.26, 312.72, -8.35) mm, rotated rx -180 ry 0 rz -179 deg; joints [9.006, -77.817, 125.426, 12.111, -48.25, -8.132]
  MoveL 169 to (-90.26, 287.32, -8.35) mm, rotated rx -180 ry 0 rz -179 deg; joints [10.214, -77.593, 125.14, 13.723, -48.372, -9.214]
  MoveL 170 to (-141.06, 287.32, -8.35) mm, rotated rx -180 ry 0 rz -179 deg; joints [10.621, -80.585, 128.864, 14.104, -49.149, -9.333]
  MoveL 171 to (-141.06, 338.12, -8.35) mm, rotated rx -180 ry 0 rz -179 deg; joints [8.094, -81.032, 129.404, 10.772, -48.877, -7.132]
  MoveL 172 to (-90.26, 338.12, -8.35) mm, rotated rx 180 ry 0 rz -179 deg; joints [7.791, -78.011, 125.672, 10.486, -48.141, -7.041]
  MoveL 173 to (-90.26, 312.72, -8.35) mm, rotated rx -180 ry 0 rz -179 deg; joints [9.006, -77.817, 125.426, 12.111, -48.25, -8.132]
  MoveC 174 to (-90.44, 312.27, -8.35) mm, rotated rx 180 ry 0 rz -179 deg; joints [9.028, -77.825, 125.435, 12.141, -48.255, -8.152] to (-90.89, 312.09, -8.35) mm, rotated rx 180 ry 0 rz -179 deg; joints [9.04, -77.849, 125.467, 12.156, -48.263, -8.16]
  MoveL 175 to (-91.53, 312.08, -8.35) mm, rotated rx -180 ry 0 rz -179 deg; joints [9.045, -77.887, 125.514, 12.159, -48.274, -8.161]
  MoveC 176 to (-91.98, 312.09, -8.16) mm, rotated rx -180 ry 0 rz -179 deg; joints [9.048, -77.921, 125.542, 12.165, -48.268, -8.166] to (-92.16, 312.08, -7.72) mm, rotated rx -180 ry 0 rz -179 deg; joints [9.049, -77.953, 125.543, 12.172, -48.238, -8.175]
  Set speed (500.0 mm/s)
  MoveL 177 to (-92.16, 312.09, 6) mm, rotated rx -180 ry 0 rz -179 deg; joints [9.049, -78.569, 125.137, 12.37, -47.239, -8.469]
  MoveL 178 to (-92.16, 499.69, 6) mm, rotated rx -180 ry 0 rz -179 deg; joints [-0.04, -79.259, 125.995, -0.054, -46.737, 0.037]
  Set speed (25.4 mm/s)
  MoveL 179 to (-92.16, 499.69, -3.54) mm, rotated rx 180 ry 0 rz -179 deg; joints [-0.04, -78.827, 126.281, -0.054, -47.454, 0.036]
  MoveC 180 to (-91.98, 499.69, -3.99) mm, rotated rx -180 ry 0 rz -179 deg; joints [-0.039, -78.795, 126.281, -0.054, -47.485, 0.036] to (-91.53, 499.69, -4.17) mm, rotated rx -180 ry 0 rz -179 deg; joints [-0.039, -78.76, 126.253, -0.053, -47.493, 0.036]
  Set speed (50.8 mm/s)
  MoveL 181 to (-90.89, 499.69, -4.18) mm, rotated rx -180 ry 0 rz -179 deg; joints [-0.039, -78.722, 126.205, -0.052, -47.483, 0.035]
  MoveC 182 to (-90.44, 499.51, -4.17) mm, rotated rx -180 ry 0 rz -179 deg; joints [-0.029, -78.696, 126.172, -0.039, -47.476, 0.027] to (-90.26, 499.06, -4.17) mm, rotated rx 180 ry 0 rz -179 deg; joints [-0.007, -78.685, 126.159, -0.01, -47.474, 0.006]
  MoveL 183 to (-90.26, 473.66, -4.18) mm, rotated rx 180 ry 0 rz -179 deg; joints [1.229, -78.695, 126.172, 1.667, -47.488, -1.126]
  MoveL 184 to (-141.06, 473.66, -4.17) mm, rotated rx -180 ry 0 rz -179 deg; joints [1.239, -81.761, 129.909, 1.663, -48.16, -1.109]
  MoveL 185 to (-141.06, 524.46, -4.18) mm, rotated rx 180 ry 0 rz -179 deg; joints [-1.343, -81.704, 129.842, -1.803, -48.152, 1.203]
  MoveL 186 to (-90.26, 524.46, -4.18) mm, rotated rx -180 ry 0 rz -179 deg; joints [-1.242, -78.642, 126.105, -1.685, -47.475, 1.139]
  MoveL 187 to (-90.26, 499.06, -4.17) mm, rotated rx 180 ry 0 rz -179 deg; joints [-0.007, -78.685, 126.159, -0.01, -47.474, 0.006]
  MoveC 188 to (-90.44, 498.61, -4.17) mm, rotated rx 180 ry 0 rz -179 deg; joints [0.015, -78.697, 126.173, 0.02, -47.477, -0.013] to (-90.89, 498.42, -4.18) mm, rotated rx -180 ry 0 rz -179 deg; joints [0.023, -78.724, 126.207, 0.032, -47.483, -0.021]
  MoveL 189 to (-91.53, 498.42, -4.17) mm, rotated rx 180 ry 0 rz -179 deg; joints [0.023, -78.761, 126.254, 0.031, -47.493, -0.021]
  MoveC 190 to (-91.98, 498.42, -3.99) mm, rotated rx -180 ry 0 rz -179 deg; joints [0.022, -78.797, 126.282, 0.03, -47.486, -0.021] to (-92.16, 498.42, -3.54) mm, rotated rx 180 ry 0 rz -179 deg; joints [0.022, -78.828, 126.283, 0.03, -47.455, -0.02]
  Set speed (500.0 mm/s)
  MoveL 191 to (-92.16, 498.42, 5) mm, rotated rx -180 ry 0 rz -179 deg; joints [0.022, -79.215, 126.027, 0.031, -46.812, -0.021]
  MoveL 192 to (-92.16, 499.69, 5) mm, rotated rx -180 ry 0 rz -179 deg; joints [-0.04, -79.214, 126.026, -0.054, -46.812, 0.037]
  Set speed (25.4 mm/s)
  MoveL 193 to (-92.16, 499.69, 1.83) mm, rotated rx 180 ry 0 rz -179 deg; joints [-0.04, -79.071, 126.121, -0.054, -47.051, 0.037]
  MoveL 194 to (-92.16, 499.69, -7.72) mm, rotated rx -180 ry 0 rz -179 deg; joints [-0.04, -78.636, 126.404, -0.054, -47.769, 0.036]
  MoveC 195 to (-91.98, 499.69, -8.16) mm, rotated rx -180 ry 0 rz -179 deg; joints [-0.039, -78.604, 126.403, -0.053, -47.8, 0.036] to (-91.53, 499.69, -8.35) mm, rotated rx 180 ry 0 rz -179 deg; joints [-0.039, -78.569, 126.375, -0.053, -47.807, 0.035]
  Set speed (50.8 mm/s)
  MoveL 196 to (-90.89, 499.69, -8.35) mm, rotated rx 180 ry 0 rz -179 deg; joints [-0.039, -78.531, 126.328, -0.052, -47.797, 0.035]
  MoveC 197 to (-90.44, 499.51, -8.35) mm, rotated rx 180 ry 0 rz -179 deg; joints [-0.029, -78.504, 126.295, -0.039, -47.79, 0.026] to (-90.26, 499.06, -8.35) mm, rotated rx -180 ry 0 rz -179 deg; joints [-0.007, -78.494, 126.281, -0.01, -47.787, 0.006]
  MoveL 198 to (-90.26, 473.66, -8.35) mm, rotated rx -180 ry 0 rz -179 deg; joints [1.229, -78.504, 126.294, 1.658, -47.802, -1.114]
  MoveL 199 to (-141.06, 473.66, -8.35) mm, rotated rx -180 ry 0 rz -179 deg; joints [1.239, -81.56, 130.036, 1.655, -48.488, -1.097]
  MoveL 200 to (-141.06, 524.46, -8.35) mm, rotated rx -180 ry 0 rz -179 deg; joints [-1.343, -81.503, 129.968, -1.793, -48.479, 1.189]
  MoveL 201 to (-90.26, 524.46, -8.35) mm, rotated rx -180 ry 0 rz -179 deg; joints [-1.242, -78.451, 126.227, -1.677, -47.789, 1.127]
  MoveL 202 to (-90.26, 499.06, -8.35) mm, rotated rx -180 ry 0 rz -179 deg; joints [-0.007, -78.494, 126.281, -0.01, -47.787, 0.006]
  MoveC 203 to (-90.44, 498.61, -8.35) mm, rotated rx -180 ry 0 rz -179 deg; joints [0.015, -78.505, 126.296, 0.02, -47.79, -0.013] to (-90.89, 498.42, -8.35) mm, rotated rx 180 ry 0 rz -179 deg; joints [0.023, -78.532, 126.329, 0.031, -47.797, -0.021]
  MoveL 204 to (-91.53, 498.42, -8.35) mm, rotated rx 180 ry 0 rz -179 deg; joints [0.023, -78.57, 126.377, 0.031, -47.807, -0.021]
  MoveC 205 to (-91.98, 498.42, -8.16) mm, rotated rx -180 ry 0 rz -179 deg; joints [0.022, -78.605, 126.405, 0.03, -47.8, -0.02] to (-92.16, 498.42, -7.72) mm, rotated rx -180 ry 0 rz -179 deg; joints [0.022, -78.637, 126.406, 0.03, -47.769, -0.02]
  Set speed (500.0 mm/s)
  MoveL 206 to (-92.16, 498.42, 6) mm, rotated rx -180 ry 0 rz -179 deg; joints [0.022, -79.26, 125.997, 0.031, -46.737, -0.021]
  MoveL 207 to (-219.16, 499.69, 6) mm, rotated rx -180 ry 0 rz -179 deg; joints [-0.165, -87.168, 135.103, -0.223, -47.935, 0.149]
  Set speed (25.4 mm/s)
  MoveL 208 to (-219.16, 499.69, -3.54) mm, rotated rx 180 ry 0 rz -179 deg; joints [-0.165, -86.68, 135.417, -0.22, -48.738, 0.145]
  MoveC 209 to (-218.98, 499.69, -3.99) mm, rotated rx -180 ry 0 rz -179 deg; joints [-0.165, -86.645, 135.419, -0.22, -48.775, 0.145] to (-218.53, 499.69, -4.17) mm, rotated rx -180 ry 0 rz -179 deg; joints [-0.165, -86.606, 135.394, -0.219, -48.788, 0.144]
  Set speed (50.8 mm/s)
  MoveL 210 to (-217.89, 499.69, -4.18) mm, rotated rx -180 ry 0 rz -179 deg; joints [-0.164, -86.565, 135.35, -0.218, -48.785, 0.144]
  MoveC 211 to (-217.44, 499.51, -4.18) mm, rotated rx -180 ry 0 rz -179 deg; joints [-0.153, -86.536, 135.319, -0.204, -48.783, 0.134] to (-217.26, 499.06, -4.18) mm, rotated rx -180 ry 0 rz -179 deg; joints [-0.129, -86.525, 135.307, -0.171, -48.782, 0.113]
  MoveL 212 to (-217.26, 473.66, -4.18) mm, rotated rx -180 ry 0 rz -179 deg; joints [1.256, -86.537, 135.32, 1.67, -48.795, -1.1]
  MoveL 213 to (-268.06, 473.66, -4.18) mm, rotated rx -180 ry 0 rz -179 deg; joints [1.269, -89.88, 138.799, 1.684, -48.932, -1.106]
  MoveL 214 to (-268.06, 524.46, -4.17) mm, rotated rx -180 ry 0 rz -179 deg; joints [-1.64, -89.809, 138.728, -2.175, -48.94, 1.429]
  MoveL 215 to (-217.26, 524.46, -4.17) mm, rotated rx -180 ry 0 rz -179 deg; joints [-1.512, -86.473, 135.25, -2.01, -48.795, 1.325]
  MoveL 216 to (-217.26, 499.06, -4.18) mm, rotated rx -180 ry 0 rz -179 deg; joints [-0.129, -86.525, 135.307, -0.171, -48.782, 0.113]
  MoveC 217 to (-217.44, 498.61, -4.18) mm, rotated rx 180 ry 0 rz -179 deg; joints [-0.104, -86.538, 135.32, -0.139, -48.783, 0.092] to (-217.89, 498.42, -4.17) mm, rotated rx -180 ry 0 rz -179 deg; joints [-0.095, -86.567, 135.352, -0.126, -48.785, 0.083]
  MoveL 218 to (-218.53, 498.42, -4.18) mm, rotated rx -180 ry 0 rz -179 deg; joints [-0.095, -86.608, 135.396, -0.127, -48.788, 0.084]
  MoveC 219 to (-218.98, 498.42, -3.99) mm, rotated rx 180 ry 0 rz -179 deg; joints [-0.096, -86.646, 135.421, -0.128, -48.775, 0.084] to (-219.16, 498.42, -3.54) mm, rotated rx -180 ry 0 rz -179 deg; joints [-0.096, -86.681, 135.419, -0.128, -48.738, 0.084]
  Set speed (500.0 mm/s)
  MoveL 220 to (-219.16, 498.42, 5) mm, rotated rx 180 ry 0 rz -179 deg; joints [-0.096, -87.119, 135.138, -0.129, -48.019, 0.086]
  MoveL 221 to (-219.16, 499.69, 5) mm, rotated rx -180 ry 0 rz -179 deg; joints [-0.165, -87.117, 135.136, -0.223, -48.019, 0.149]
  Set speed (25.4 mm/s)
  MoveL 222 to (-219.16, 499.69, 1.82) mm, rotated rx -180 ry 0 rz -179 deg; joints [-0.165, -86.956, 135.241, -0.222, -48.286, 0.148]
  MoveL 223 to (-219.16, 499.69, -7.72) mm, rotated rx -180 ry 0 rz -179 deg; joints [-0.165, -86.463, 135.552, -0.219, -49.09, 0.143]
  MoveC 224 to (-218.98, 499.69, -8.16) mm, rotated rx -180 ry 0 rz -179 deg; joints [-0.165, -86.427, 135.554, -0.219, -49.127, 0.143] to (-218.53, 499.69, -8.35) mm, rotated rx -180 ry 0 rz -179 deg; joints [-0.165, -86.389, 135.529, -0.218, -49.14, 0.143]
  Set speed (50.8 mm/s)
  MoveL 225 to (-217.89, 499.69, -8.35) mm, rotated rx 180 ry 0 rz -179 deg; joints [-0.164, -86.348, 135.485, -0.217, -49.137, 0.142]
  MoveC 226 to (-217.44, 499.51, -8.35) mm, rotated rx 180 ry 0 rz -179 deg; joints [-0.153, -86.32, 135.454, -0.203, -49.134, 0.133] to (-217.26, 499.06, -8.35) mm, rotated rx -180 ry 0 rz -179 deg; joints [-0.129, -86.308, 135.441, -0.17, -49.133, 0.111]
  MoveL 227 to (-217.26, 473.66, -8.35) mm, rotated rx 180 ry 0 rz -179 deg; joints [1.256, -86.321, 135.455, 1.661, -49.146, -1.087]
  MoveL 228 to (-268.06, 473.66, -8.35) mm, rotated rx 180 ry 0 rz -179 deg; joints [1.269, -89.652, 138.94, 1.674, -49.3, -1.092]
  MoveL 229 to (-268.06, 524.46, -8.35) mm, rotated rx -180 ry 0 rz -179 deg; joints [-1.64, -89.581, 138.869, -2.163, -49.308, 1.411]
  MoveL 230 to (-217.26, 524.46, -8.35) mm, rotated rx 180 ry 0 rz -179 deg; joints [-1.512, -86.256, 135.385, -2, -49.146, 1.308]
  MoveL 231 to (-217.26, 499.06, -8.35) mm, rotated rx -180 ry 0 rz -179 deg; joints [-0.129, -86.308, 135.441, -0.17, -49.133, 0.111]
  MoveC 232 to (-217.44, 498.61, -8.35) mm, rotated rx -180 ry 0 rz -179 deg; joints [-0.104, -86.321, 135.455, -0.138, -49.134, 0.09] to (-217.89, 498.42, -8.35) mm, rotated rx -180 ry 0 rz -179 deg; joints [-0.095, -86.35, 135.486, -0.125, -49.137, 0.082]
  MoveL 233 to (-218.53, 498.42, -8.35) mm, rotated rx -180 ry 0 rz -179 deg; joints [-0.095, -86.391, 135.53, -0.126, -49.14, 0.083]
  MoveC 234 to (-218.98, 498.42, -8.16) mm, rotated rx -180 ry 0 rz -179 deg; joints [-0.096, -86.429, 135.556, -0.127, -49.127, 0.083] to (-219.16, 498.42, -7.72) mm, rotated rx -180 ry 0 rz -179 deg; joints [-0.096, -86.464, 135.554, -0.127, -49.09, 0.083]
  Set speed (500.0 mm/s)
  MoveL 235 to (-219.16, 498.42, 6) mm, rotated rx -180 ry 0 rz -179 deg; joints [-0.096, -87.169, 135.105, -0.129, -47.935, 0.087]
  MoveL 236 to (-346.16, 499.69, 6) mm, rotated rx -180 ry 0 rz -179 deg; joints [-0.326, -95.921, 143.551, -0.441, -47.632, 0.297]
  Set speed (25.4 mm/s)
  MoveL 237 to (-346.16, 499.69, -3.54) mm, rotated rx -180 ry 0 rz -179 deg; joints [-0.326, -95.372, 143.907, -0.435, -48.535, 0.288]
  MoveC 238 to (-345.98, 499.69, -3.99) mm, rotated rx -180 ry 0 rz -179 deg; joints [-0.326, -95.333, 143.911, -0.434, -48.58, 0.287] to (-345.53, 499.69, -4.17) mm, rotated rx 180 ry 0 rz -179 deg; joints [-0.325, -95.289, 143.889, -0.433, -48.601, 0.287]
  Set speed (50.8 mm/s)
  MoveL 239 to (-344.89, 499.69, -4.17) mm, rotated rx -180 ry 0 rz -179 deg; joints [-0.324, -95.243, 143.848, -0.432, -48.607, 0.286]
  MoveC 240 to (-344.44, 499.51, -4.17) mm, rotated rx 180 ry 0 rz -179 deg; joints [-0.312, -95.21, 143.82, -0.416, -48.611, 0.275] to (-344.26, 499.06, -4.18) mm, rotated rx -180 ry 0 rz -179 deg; joints [-0.284, -95.197, 143.809, -0.378, -48.612, 0.25]
  MoveL 241 to (-344.26, 473.66, -4.17) mm, rotated rx -180 ry 0 rz -179 deg; joints [1.291, -95.213, 143.823, 1.721, -48.622, -1.138]
  MoveL 242 to (-395.06, 473.66, -4.17) mm, rotated rx 180 ry 0 rz -179 deg; joints [1.308, -99.043, 147.034, 1.761, -48.005, -1.178]
  MoveL 243 to (-395.06, 524.46, -4.18) mm, rotated rx -180 ry 0 rz -179 deg; joints [-2.023, -98.949, 146.96, -2.721, -48.043, 1.82]
  MoveL 244 to (-344.26, 524.46, -4.17) mm, rotated rx 180 ry 0 rz -179 deg; joints [-1.857, -95.13, 143.749, -2.475, -48.646, 1.636]
  MoveL 245 to (-344.26, 499.06, -4.18) mm, rotated rx -180 ry 0 rz -179 deg; joints [-0.284, -95.197, 143.809, -0.378, -48.612, 0.25]
  MoveC 246 to (-344.44, 498.61, -4.17) mm, rotated rx 180 ry 0 rz -179 deg; joints [-0.256, -95.212, 143.821, -0.342, -48.61, 0.226] to (-344.89, 498.42, -4.18) mm, rotated rx -180 ry 0 rz -179 deg; joints [-0.245, -95.245, 143.85, -0.327, -48.606, 0.216]
  MoveL 247 to (-345.53, 498.42, -4.17) mm, rotated rx -180 ry 0 rz -179 deg; joints [-0.246, -95.291, 143.891, -0.328, -48.601, 0.217]
  MoveC 248 to (-345.98, 498.42, -3.99) mm, rotated rx 180 ry 0 rz -179 deg; joints [-0.247, -95.335, 143.913, -0.329, -48.579, 0.218] to (-346.16, 498.42, -3.54) mm, rotated rx -180 ry 0 rz -179 deg; joints [-0.247, -95.374, 143.909, -0.33, -48.535, 0.218]
  Set speed (500.0 mm/s)
  MoveL 249 to (-346.16, 498.42, 5) mm, rotated rx 180 ry 0 rz -179 deg; joints [-0.247, -95.866, 143.591, -0.334, -47.725, 0.225]
  MoveL 250 to (-346.16, 499.69, 5) mm, rotated rx -180 ry 0 rz -179 deg; joints [-0.326, -95.864, 143.589, -0.441, -47.726, 0.296]
  Set speed (25.4 mm/s)
  MoveL 251 to (-346.16, 499.69, 1.83) mm, rotated rx -180 ry 0 rz -179 deg; joints [-0.326, -95.682, 143.708, -0.438, -48.026, 0.293]
  MoveL 252 to (-346.16, 499.69, -7.71) mm, rotated rx 180 ry 0 rz -179 deg; joints [-0.326, -95.128, 144.06, -0.432, -48.933, 0.284]
  MoveC 253 to (-345.98, 499.69, -8.16) mm, rotated rx 180 ry 0 rz -179 deg; joints [-0.326, -95.088, 144.064, -0.432, -48.977, 0.283] to (-345.53, 499.69, -8.35) mm, rotated rx 180 ry 0 rz -179 deg; joints [-0.325, -95.044, 144.042, -0.431, -48.998, 0.283]
  Set speed (50.8 mm/s)
  MoveL 254 to (-344.89, 499.69, -8.35) mm, rotated rx -180 ry 0 rz -179 deg; joints [-0.324, -94.998, 144.001, -0.43, -49.004, 0.282]
  MoveC 255 to (-344.44, 499.51, -8.35) mm, rotated rx -180 ry 0 rz -179 deg; joints [-0.312, -94.966, 143.972, -0.413, -49.007, 0.271] to (-344.26, 499.06, -8.35) mm, rotated rx 180 ry 0 rz -179 deg; joints [-0.284, -94.953, 143.961, -0.376, -49.009, 0.247]
  MoveL 256 to (-344.26, 473.66, -8.35) mm, rotated rx 180 ry 0 rz -179 deg; joints [1.291, -94.969, 143.975, 1.711, -49.019, -1.122]
  MoveL 257 to (-395.06, 473.66, -8.35) mm, rotated rx 180 ry 0 rz -179 deg; joints [1.308, -98.787, 147.196, 1.749, -48.422, -1.161]
  MoveL 258 to (-395.06, 524.46, -8.35) mm, rotated rx -180 ry 0 rz -179 deg; joints [-2.023, -98.694, 147.121, -2.704, -48.459, 1.794]
  MoveL 259 to (-344.26, 524.46, -8.35) mm, rotated rx -180 ry 0 rz -179 deg; joints [-1.857, -94.886, 143.902, -2.46, -49.042, 1.613]
  MoveL 260 to (-344.26, 499.06, -8.35) mm, rotated rx 180 ry 0 rz -179 deg; joints [-0.284, -94.953, 143.961, -0.376, -49.009, 0.247]
  MoveC 261 to (-344.44, 498.61, -8.35) mm, rotated rx 180 ry 0 rz -179 deg; joints [-0.256, -94.967, 143.974, -0.34, -49.007, 0.223] to (-344.89, 498.42, -8.35) mm, rotated rx -180 ry 0 rz -179 deg; joints [-0.245, -95, 144.003, -0.325, -49.003, 0.213]
  MoveL 262 to (-345.53, 498.42, -8.35) mm, rotated rx -180 ry 0 rz -179 deg; joints [-0.246, -95.046, 144.044, -0.326, -48.998, 0.214]
  MoveC 263 to (-345.98, 498.42, -8.16) mm, rotated rx -180 ry 0 rz -179 deg; joints [-0.247, -95.09, 144.066, -0.327, -48.976, 0.215] to (-346.16, 498.42, -7.72) mm, rotated rx -180 ry 0 rz -179 deg; joints [-0.247, -95.13, 144.061, -0.328, -48.932, 0.215]
  Set speed (500.0 mm/s)
  MoveL 264 to (-346.16, 498.42, 6) mm, rotated rx -180 ry 0 rz -179 deg; joints [-0.247, -95.923, 143.553, -0.334, -47.631, 0.225]
  MoveL 265 to (139.15, 499.69, 6) mm, rotated rx -180 ry 0 rz -179 deg; joints [0.131, -65.766, 107.508, 0.197, -41.742, -0.147]
  Set speed (25.4 mm/s)
  MoveL 266 to (139.15, 499.69, -3.54) mm, rotated rx -180 ry 0 rz -179 deg; joints [0.131, -65.422, 107.767, 0.195, -42.345, -0.144]
  MoveC 267 to (139.34, 499.69, -3.99) mm, rotated rx -180 ry 0 rz -179 deg; joints [0.131, -65.395, 107.763, 0.195, -42.368, -0.144] to (139.79, 499.69, -4.17) mm, rotated rx -180 ry 0 rz -179 deg; joints [0.132, -65.362, 107.729, 0.195, -42.367, -0.144]
  Set speed (50.8 mm/s)
  MoveL 268 to (140.42, 499.69, -4.17) mm, rotated rx -180 ry 0 rz -179 deg; joints [0.132, -65.326, 107.674, 0.196, -42.348, -0.145]
  MoveC 269 to (140.87, 499.51, -4.17) mm, rotated rx -180 ry 0 rz -179 deg; joints [0.14, -65.3, 107.635, 0.208, -42.335, -0.154] to (141.06, 499.06, -4.17) mm, rotated rx 180 ry 0 rz -179 deg; joints [0.158, -65.29, 107.62, 0.235, -42.33, -0.174]
  MoveL 270 to (141.06, 473.66, -4.18) mm, rotated rx -180 ry 0 rz -179 deg; joints [1.191, -65.298, 107.632, 1.768, -42.348, -1.307]
  MoveL 271 to (90.26, 473.66, -4.17) mm, rotated rx -180 ry 0 rz -179 deg; joints [1.198, -68.212, 111.946, 1.733, -43.747, -1.252]
  MoveL 272 to (90.26, 524.46, -4.18) mm, rotated rx 180 ry 0 rz -179 deg; joints [-0.944, -68.168, 111.882, -1.366, -43.722, 0.987]
  MoveL 273 to (141.06, 524.46, -4.18) mm, rotated rx 180 ry 0 rz -179 deg; joints [-0.874, -65.255, 107.568, -1.298, -42.32, 0.96]
  MoveL 274 to (141.06, 499.06, -4.17) mm, rotated rx 180 ry 0 rz -179 deg; joints [0.158, -65.29, 107.62, 0.235, -42.33, -0.174]
  MoveC 275 to (140.87, 498.61, -4.17) mm, rotated rx -180 ry 0 rz -179 deg; joints [0.176, -65.301, 107.637, 0.262, -42.336, -0.194] to (140.42, 498.42, -4.18) mm, rotated rx 180 ry 0 rz -179 deg; joints [0.184, -65.327, 107.676, 0.273, -42.349, -0.202]
  MoveL 276 to (139.79, 498.42, -4.17) mm, rotated rx 180 ry 0 rz -179 deg; joints [0.183, -65.363, 107.73, 0.272, -42.367, -0.201]
  MoveC 277 to (139.34, 498.42, -3.99) mm, rotated rx 180 ry 0 rz -179 deg; joints [0.183, -65.396, 107.764, 0.272, -42.369, -0.201] to (139.15, 498.42, -3.54) mm, rotated rx 180 ry 0 rz -179 deg; joints [0.183, -65.423, 107.768, 0.272, -42.346, -0.201]
  Set speed (500.0 mm/s)
  MoveL 278 to (139.15, 498.42, 5) mm, rotated rx -180 ry 0 rz -179 deg; joints [0.183, -65.731, 107.537, 0.274, -41.806, -0.205]
  MoveL 279 to (139.15, 499.69, 5) mm, rotated rx -180 ry 0 rz -179 deg; joints [0.131, -65.73, 107.535, 0.197, -41.805, -0.147]
  Set speed (25.4 mm/s)
  MoveL 280 to (139.15, 499.69, 1.82) mm, rotated rx -180 ry 0 rz -179 deg; joints [0.131, -65.616, 107.622, 0.196, -42.006, -0.146]
  MoveL 281 to (139.15, 499.69, -7.72) mm, rotated rx -180 ry 0 rz -179 deg; joints [0.131, -65.269, 107.878, 0.194, -42.609, -0.143]
  MoveC 282 to (139.34, 499.69, -8.16) mm, rotated rx -180 ry 0 rz -179 deg; joints [0.131, -65.242, 107.874, 0.194, -42.631, -0.143] to (139.79, 499.69, -8.35) mm, rotated rx -180 ry 0 rz -179 deg; joints [0.132, -65.21, 107.84, 0.194, -42.63, -0.143]
  Set speed (50.8 mm/s)
  MoveL 283 to (140.42, 499.69, -8.35) mm, rotated rx -180 ry 0 rz -179 deg; joints [0.132, -65.173, 107.785, 0.195, -42.612, -0.144]
  MoveC 284 to (140.87, 499.51, -8.35) mm, rotated rx 180 ry 0 rz -179 deg; joints [0.14, -65.148, 107.746, 0.207, -42.599, -0.152] to (141.06, 499.06, -8.35) mm, rotated rx 180 ry 0 rz -179 deg; joints [0.158, -65.138, 107.731, 0.234, -42.593, -0.172]
  MoveL 285 to (141.06, 473.66, -8.35) mm, rotated rx -180 ry 0 rz -179 deg; joints [1.191, -65.146, 107.743, 1.759, -42.611, -1.295]
  MoveL 286 to (90.26, 473.66, -8.35) mm, rotated rx 180 ry 0 rz -179 deg; joints [1.198, -68.052, 112.059, 1.724, -44.019, -1.24]
  MoveL 287 to (90.26, 524.46, -8.35) mm, rotated rx -180 ry 0 rz -179 deg; joints [-0.944, -68.008, 111.994, -1.359, -43.994, 0.978]
  MoveL 288 to (141.06, 524.46, -8.35) mm, rotated rx 180 ry 0 rz -179 deg; joints [-0.874, -65.103, 107.679, -1.292, -42.583, 0.951]
  MoveL 289 to (141.06, 499.06, -8.35) mm, rotated rx 180 ry 0 rz -179 deg; joints [0.158, -65.138, 107.731, 0.234, -42.593, -0.172]
  MoveC 290 to (140.87, 498.61, -8.35) mm, rotated rx 180 ry 0 rz -179 deg; joints [0.176, -65.149, 107.747, 0.261, -42.599, -0.192] to (140.42, 498.42, -8.35) mm, rotated rx -180 ry 0 rz -179 deg; joints [0.184, -65.174, 107.786, 0.271, -42.612, -0.2]
  MoveL 291 to (139.79, 498.42, -8.35) mm, rotated rx 180 ry 0 rz -179 deg; joints [0.183, -65.211, 107.841, 0.271, -42.631, -0.199]
  MoveC 292 to (139.34, 498.42, -8.16) mm, rotated rx -180 ry 0 rz -179 deg; joints [0.183, -65.243, 107.875, 0.27, -42.632, -0.199] to (139.15, 498.42, -7.72) mm, rotated rx -180 ry 0 rz -179 deg; joints [0.183, -65.271, 107.879, 0.27, -42.609, -0.199]
  Set speed (500.0 mm/s)
  MoveL 293 to (139.15, 498.42, 6) mm, rotated rx -180 ry 0 rz -179 deg; joints [0.183, -65.767, 107.509, 0.275, -41.743, -0.205]
  MoveL 294 to (266.15, 499.69, 6) mm, rotated rx -180 ry 0 rz -179 deg; joints [0.203, -58.319, 95.962, 0.333, -37.643, -0.263]
  Set speed (25.4 mm/s)
  MoveL 295 to (266.15, 499.69, -3.54) mm, rotated rx -180 ry 0 rz -179 deg; joints [0.203, -58.018, 96.22, 0.328, -38.202, -0.258]
  MoveC 296 to (266.34, 499.69, -3.99) mm, rotated rx 180 ry 0 rz -179 deg; joints [0.203, -57.992, 96.214, 0.329, -38.222, -0.258] to (266.79, 499.69, -4.17) mm, rotated rx 180 ry 0 rz -179 deg; joints [0.203, -57.96, 96.176, 0.329, -38.216, -0.258]
  Set speed (50.8 mm/s)
  MoveL 297 to (267.42, 499.69, -4.17) mm, rotated rx -180 ry 0 rz -179 deg; joints [0.204, -57.922, 96.115, 0.33, -38.193, -0.259]
  MoveC 298 to (267.87, 499.51, -4.18) mm, rotated rx 180 ry 0 rz -179 deg; joints [0.211, -57.895, 96.072, 0.341, -38.177, -0.268] to (268.06, 499.06, -4.18) mm, rotated rx -180 ry 0 rz -179 deg; joints [0.228, -57.885, 96.054, 0.369, -38.17, -0.29]
  MoveL 299 to (268.06, 473.66, -4.18) mm, rotated rx -180 ry 0 rz -179 deg; joints [1.175, -57.893, 96.067, 1.901, -38.19, -1.494]
  MoveL 300 to (217.26, 473.66, -4.17) mm, rotated rx 180 ry 0 rz -179 deg; joints [1.181, -60.888, 100.843, 1.839, -39.97, -1.41]
  MoveL 301 to (217.26, 524.46, -4.17) mm, rotated rx 180 ry 0 rz -179 deg; joints [-0.778, -60.846, 100.778, -1.212, -39.938, 0.929]
  MoveL 302 to (268.06, 524.46, -4.18) mm, rotated rx -180 ry 0 rz -179 deg; joints [-0.719, -57.852, 96.001, -1.164, -38.155, 0.915]
  MoveL 303 to (268.06, 499.06, -4.18) mm, rotated rx -180 ry 0 rz -179 deg; joints [0.228, -57.885, 96.054, 0.369, -38.17, -0.29]
  MoveC 304 to (267.87, 498.61, -4.18) mm, rotated rx -180 ry 0 rz -179 deg; joints [0.244, -57.896, 96.073, 0.396, -38.177, -0.311] to (267.42, 498.42, -4.18) mm, rotated rx 180 ry 0 rz -179 deg; joints [0.251, -57.923, 96.116, 0.406, -38.194, -0.319]
  MoveL 305 to (266.79, 498.42, -4.17) mm, rotated rx -180 ry 0 rz -179 deg; joints [0.251, -57.961, 96.177, 0.406, -38.217, -0.319]
  MoveC 306 to (266.34, 498.42, -3.99) mm, rotated rx 180 ry 0 rz -179 deg; joints [0.251, -57.993, 96.215, 0.405, -38.223, -0.318] to (266.15, 498.42, -3.54) mm, rotated rx -180 ry 0 rz -179 deg; joints [0.251, -58.019, 96.221, 0.405, -38.203, -0.318]
  Set speed (500.0 mm/s)
  MoveL 307 to (266.15, 498.42, 5) mm, rotated rx -180 ry 0 rz -179 deg; joints [0.251, -58.289, 95.991, 0.41, -37.703, -0.324]
  MoveL 308 to (266.15, 499.69, 5) mm, rotated rx -180 ry 0 rz -179 deg; joints [0.203, -58.288, 95.99, 0.332, -37.702, -0.263]
  Set speed (25.4 mm/s)
  MoveL 309 to (266.15, 499.69, 1.83) mm, rotated rx 180 ry 0 rz -179 deg; joints [0.203, -58.188, 96.076, 0.331, -37.888, -0.261]
  MoveL 310 to (266.15, 499.69, -7.72) mm, rotated rx -180 ry 0 rz -179 deg; joints [0.203, -57.884, 96.33, 0.327, -38.446, -0.256]
  MoveC 311 to (266.34, 499.69, -8.16) mm, rotated rx -180 ry 0 rz -179 deg; joints [0.203, -57.859, 96.324, 0.327, -38.466, -0.256] to (266.79, 499.69, -8.35) mm, rotated rx 180 ry 0 rz -179 deg; joints [0.203, -57.826, 96.286, 0.327, -38.46, -0.256]
  Set speed (50.8 mm/s)
  MoveL 312 to (267.42, 499.69, -8.35) mm, rotated rx -180 ry 0 rz -179 deg; joints [0.204, -57.788, 96.225, 0.328, -38.437, -0.257]
  MoveC 313 to (267.87, 499.51, -8.35) mm, rotated rx -180 ry 0 rz -179 deg; joints [0.211, -57.762, 96.182, 0.34, -38.42, -0.266] to (268.06, 499.06, -8.35) mm, rotated rx -180 ry 0 rz -179 deg; joints [0.228, -57.751, 96.164, 0.367, -38.414, -0.287]
  MoveL 314 to (268.06, 473.66, -8.35) mm, rotated rx 180 ry 0 rz -179 deg; joints [1.175, -57.759, 96.177, 1.891, -38.433, -1.481]
  MoveL 315 to (217.26, 473.66, -8.35) mm, rotated rx 180 ry 0 rz -179 deg; joints [1.181, -60.747, 100.953, 1.829, -40.22, -1.397]
  MoveL 316 to (217.26, 524.46, -8.35) mm, rotated rx -180 ry 0 rz -179 deg; joints [-0.778, -60.706, 100.888, -1.206, -40.188, 0.921]
  MoveL 317 to (268.06, 524.46, -8.35) mm, rotated rx -180 ry 0 rz -179 deg; joints [-0.719, -57.718, 96.111, -1.158, -38.399, 0.907]
  MoveL 318 to (268.06, 499.06, -8.35) mm, rotated rx -180 ry 0 rz -179 deg; joints [0.228, -57.751, 96.164, 0.367, -38.414, -0.287]
  MoveC 319 to (267.87, 498.61, -8.35) mm, rotated rx -180 ry 0 rz -179 deg; joints [0.244, -57.762, 96.183, 0.393, -38.421, -0.308] to (267.42, 498.42, -8.35) mm, rotated rx -180 ry 0 rz -179 deg; joints [0.251, -57.789, 96.226, 0.404, -38.438, -0.317]
  MoveL 320 to (266.79, 498.42, -8.35) mm, rotated rx -180 ry 0 rz -179 deg; joints [0.251, -57.827, 96.287, 0.403, -38.461, -0.316]
  MoveC 321 to (266.34, 498.42, -8.16) mm, rotated rx 180 ry 0 rz -179 deg; joints [0.251, -57.86, 96.326, 0.403, -38.467, -0.316] to (266.15, 498.42, -7.72) mm, rotated rx 180 ry 0 rz -179 deg; joints [0.251, -57.885, 96.332, 0.403, -38.447, -0.316]
  Set speed (500.0 mm/s)
  MoveL 322 to (266.15, 498.42, 6) mm, rotated rx 180 ry 0 rz -179 deg; joints [0.251, -58.32, 95.964, 0.41, -37.644, -0.325]
  MoveL 323 to (393.15, 499.69, 6) mm, rotated rx 180 ry 0 rz -179 deg; joints [0.264, -50.422, 82.885, 0.492, -32.464, -0.415]
  Set speed (25.4 mm/s)
  MoveL 324 to (393.15, 499.69, -3.54) mm, rotated rx 180 ry 0 rz -179 deg; joints [0.264, -50.163, 83.153, 0.485, -32.992, -0.407]
  MoveC 325 to (393.34, 499.69, -3.99) mm, rotated rx -180 ry 0 rz -179 deg; joints [0.264, -50.138, 83.145, 0.485, -33.008, -0.407] to (393.79, 499.69, -4.17) mm, rotated rx 180 ry 0 rz -179 deg; joints [0.264, -50.104, 83.101, 0.485, -32.998, -0.407]
  Set speed (50.8 mm/s)
  MoveL 326 to (394.42, 499.69, -4.17) mm, rotated rx -180 ry 0 rz -179 deg; joints [0.265, -50.063, 83.03, 0.486, -32.968, -0.408]
  MoveC 327 to (394.87, 499.51, -4.17) mm, rotated rx 180 ry 0 rz -179 deg; joints [0.271, -50.034, 82.98, 0.499, -32.948, -0.419] to (395.06, 499.06, -4.18) mm, rotated rx 180 ry 0 rz -179 deg; joints [0.287, -50.022, 82.96, 0.527, -32.939, -0.443]
  MoveL 328 to (395.06, 473.66, -4.18) mm, rotated rx -180 ry 0 rz -179 deg; joints [1.162, -50.03, 82.974, 2.136, -32.962, -1.792]
  MoveL 329 to (344.26, 473.66, -4.17) mm, rotated rx -180 ry 0 rz -179 deg; joints [1.167, -53.258, 88.441, 2.025, -35.2, -1.655]
  MoveL 330 to (344.26, 524.46, -4.17) mm, rotated rx -180 ry 0 rz -179 deg; joints [-0.638, -53.217, 88.373, -1.108, -35.16, 0.906]
  MoveL 331 to (395.06, 524.46, -4.17) mm, rotated rx -180 ry 0 rz -179 deg; joints [-0.588, -49.989, 82.904, -1.082, -32.919, 0.908]
  MoveL 332 to (395.06, 499.06, -4.18) mm, rotated rx 180 ry 0 rz -179 deg; joints [0.287, -50.022, 82.96, 0.527, -32.939, -0.443]
  MoveC 333 to (394.87, 498.61, -4.17) mm, rotated rx -180 ry 0 rz -179 deg; joints [0.302, -50.034, 82.982, 0.556, -32.948, -0.466] to (394.42, 498.42, -4.17) mm, rotated rx 180 ry 0 rz -179 deg; joints [0.308, -50.064, 83.032, 0.567, -32.969, -0.475]
  MoveL 334 to (393.79, 498.42, -4.18) mm, rotated rx 180 ry 0 rz -179 deg; joints [0.308, -50.105, 83.102, 0.566, -32.999, -0.475]
  MoveC 335 to (393.34, 498.42, -3.99) mm, rotated rx -180 ry 0 rz -179 deg; joints [0.308, -50.139, 83.147, 0.565, -33.009, -0.474] to (393.15, 498.42, -3.54) mm, rotated rx -180 ry 0 rz -179 deg; joints [0.308, -50.164, 83.155, 0.565, -32.993, -0.474]
  Set speed (500.0 mm/s)
  MoveL 336 to (393.15, 498.42, 5) mm, rotated rx 180 ry 0 rz -179 deg; joints [0.308, -50.396, 82.915, 0.573, -32.52, -0.483]
  MoveL 337 to (393.15, 499.69, 5) mm, rotated rx -180 ry 0 rz -179 deg; joints [0.264, -50.395, 82.913, 0.491, -32.519, -0.414]
  Set speed (25.4 mm/s)
  MoveL 338 to (393.15, 499.69, 1.82) mm, rotated rx -180 ry 0 rz -179 deg; joints [0.264, -50.309, 83.003, 0.489, -32.695, -0.411]
  MoveL 339 to (393.15, 499.69, -7.72) mm, rotated rx -180 ry 0 rz -179 deg; joints [0.264, -50.047, 83.268, 0.482, -33.222, -0.403]
  MoveC 340 to (393.34, 499.69, -8.16) mm, rotated rx 180 ry 0 rz -179 deg; joints [0.264, -50.023, 83.26, 0.482, -33.238, -0.403] to (393.79, 499.69, -8.35) mm, rotated rx 180 ry 0 rz -179 deg; joints [0.264, -49.989, 83.215, 0.482, -33.228, -0.404]
  Set speed (50.8 mm/s)
  MoveL 341 to (394.42, 499.69, -8.35) mm, rotated rx -180 ry 0 rz -179 deg; joints [0.265, -49.947, 83.145, 0.483, -33.198, -0.404]
  MoveC 342 to (394.87, 499.51, -8.35) mm, rotated rx 180 ry 0 rz -179 deg; joints [0.271, -49.919, 83.095, 0.496, -33.178, -0.415] to (395.06, 499.06, -8.35) mm, rotated rx -180 ry 0 rz -179 deg; joints [0.287, -49.907, 83.075, 0.524, -33.169, -0.439]
  MoveL 343 to (395.06, 473.66, -8.35) mm, rotated rx -180 ry 0 rz -179 deg; joints [1.162, -49.915, 83.089, 2.123, -33.192, -1.777]
  MoveL 344 to (344.26, 473.66, -8.35) mm, rotated rx 180 ry 0 rz -179 deg; joints [1.167, -53.135, 88.553, 2.013, -35.434, -1.64]
  MoveL 345 to (344.26, 524.46, -8.35) mm, rotated rx -180 ry 0 rz -179 deg; joints [-0.638, -53.095, 88.485, -1.101, -35.395, 0.898]
  MoveL 346 to (395.06, 524.46, -8.35) mm, rotated rx -180 ry 0 rz -179 deg; joints [-0.588, -49.874, 83.019, -1.075, -33.149, 0.9]
  MoveL 347 to (395.06, 499.06, -8.35) mm, rotated rx -180 ry 0 rz -179 deg; joints [0.287, -49.907, 83.075, 0.524, -33.169, -0.439]
  MoveC 348 to (394.87, 498.61, -8.35) mm, rotated rx -180 ry 0 rz -179 deg; joints [0.302, -49.919, 83.096, 0.552, -33.178, -0.462] to (394.42, 498.42, -8.35) mm, rotated rx -180 ry 0 rz -179 deg; joints [0.308, -49.949, 83.147, 0.563, -33.199, -0.471]
  MoveL 349 to (393.79, 498.42, -8.35) mm, rotated rx -180 ry 0 rz -179 deg; joints [0.308, -49.99, 83.217, 0.562, -33.229, -0.47]
  MoveC 350 to (393.34, 498.42, -8.16) mm, rotated rx -180 ry 0 rz -179 deg; joints [0.308, -50.024, 83.262, 0.562, -33.239, -0.47] to (393.15, 498.42, -7.72) mm, rotated rx -180 ry 0 rz -179 deg; joints [0.308, -50.048, 83.27, 0.562, -33.223, -0.47]
  Set speed (500.0 mm/s)
  MoveL 351 to (393.15, 498.42, 6) mm, rotated rx -180 ry 0 rz -179 deg; joints [0.308, -50.423, 82.887, 0.574, -32.465, -0.484]
  MoveL 352 to (393.15, 313.36, 6) mm, rotated rx 180 ry 0 rz -179 deg; joints [6.673, -49.896, 81.987, 12.419, -32.705, -10.498]
  Set speed (25.4 mm/s)
  MoveL 353 to (393.15, 313.36, -3.54) mm, rotated rx -180 ry 0 rz -179 deg; joints [6.673, -49.639, 82.257, 12.245, -33.219, -10.291]
  MoveC 354 to (393.34, 313.36, -3.99) mm, rotated rx -180 ry 0 rz -179 deg; joints [6.672, -49.615, 82.249, 12.239, -33.235, -10.284] to (393.79, 313.36, -4.17) mm, rotated rx -180 ry 0 rz -179 deg; joints [6.671, -49.581, 82.204, 12.24, -33.224, -10.286]
  Set speed (50.8 mm/s)
  MoveL 355 to (394.42, 313.36, -4.17) mm, rotated rx -180 ry 0 rz -179 deg; joints [6.668, -49.539, 82.133, 12.246, -33.195, -10.294]
  MoveC 356 to (394.87, 313.17, -4.18) mm, rotated rx -180 ry 0 rz -179 deg; joints [6.673, -49.509, 82.08, 12.261, -33.174, -10.31] to (395.06, 312.72, -4.18) mm, rotated rx 180 ry 0 rz -179 deg; joints [6.688, -49.494, 82.055, 12.291, -33.166, -10.336]
  MoveL 357 to (395.06, 287.32, -4.17) mm, rotated rx -180 ry 0 rz -179 deg; joints [7.553, -49.316, 81.75, 13.887, -33.207, -11.687]
  MoveL 358 to (344.26, 287.32, -4.17) mm, rotated rx -180 ry 0 rz -179 deg; joints [7.758, -52.553, 87.257, 13.457, -35.454, -11.029]
  MoveL 359 to (344.26, 338.12, -4.18) mm, rotated rx -180 ry 0 rz -179 deg; joints [5.971, -52.878, 87.804, 10.354, -35.369, -8.474]
  MoveL 360 to (395.06, 338.12, -4.17) mm, rotated rx 180 ry 0 rz -179 deg; joints [5.82, -49.646, 82.316, 10.693, -33.128, -8.986]
  MoveL 361 to (395.06, 312.72, -4.18) mm, rotated rx 180 ry 0 rz -179 deg; joints [6.688, -49.494, 82.055, 12.291, -33.166, -10.336]
  MoveC 362 to (394.87, 312.27, -4.17) mm, rotated rx -180 ry 0 rz -179 deg; joints [6.704, -49.503, 82.07, 12.318, -33.176, -10.357] to (394.42, 312.09, -4.18) mm, rotated rx -180 ry 0 rz -179 deg; joints [6.712, -49.531, 82.119, 12.325, -33.197, -10.361]
  MoveL 363 to (393.79, 312.09, -4.17) mm, rotated rx -180 ry 0 rz -179 deg; joints [6.714, -49.572, 82.19, 12.32, -33.226, -10.353]
  MoveC 364 to (393.34, 312.09, -3.99) mm, rotated rx -180 ry 0 rz -179 deg; joints [6.715, -49.607, 82.235, 12.319, -33.237, -10.351] to (393.15, 312.09, -3.54) mm, rotated rx -180 ry 0 rz -179 deg; joints [6.716, -49.631, 82.243, 12.325, -33.221, -10.358]
  Set speed (500.0 mm/s)
  MoveL 365 to (393.15, 312.09, 5) mm, rotated rx -180 ry 0 rz -179 deg; joints [6.716, -49.861, 82.002, 12.481, -32.761, -10.544]
  MoveL 366 to (393.15, 313.36, 5) mm, rotated rx -180 ry 0 rz -179 deg; joints [6.673, -49.869, 82.016, 12.4, -32.759, -10.476]
  Set speed (25.4 mm/s)
  MoveL 367 to (393.15, 313.36, 1.82) mm, rotated rx -180 ry 0 rz -179 deg; joints [6.673, -49.784, 82.106, 12.342, -32.93, -10.406]
  MoveL 368 to (393.15, 313.36, -7.72) mm, rotated rx -180 ry 0 rz -179 deg; joints [6.673, -49.525, 82.372, 12.172, -33.444, -10.203]
  MoveC 369 to (393.34, 313.36, -8.16) mm, rotated rx 180 ry 0 rz -179 deg; joints [6.672, -49.501, 82.364, 12.165, -33.459, -10.196] to (393.79, 313.36, -8.35) mm, rotated rx 180 ry 0 rz -179 deg; joints [6.671, -49.467, 82.319, 12.166, -33.448, -10.197]
  Set speed (50.8 mm/s)
  MoveL 370 to (394.42, 313.36, -8.35) mm, rotated rx 180 ry 0 rz -179 deg; joints [6.668, -49.425, 82.248, 12.172, -33.419, -10.206]
  MoveC 371 to (394.87, 313.17, -8.35) mm, rotated rx -180 ry 0 rz -179 deg; joints [6.673, -49.395, 82.196, 12.187, -33.398, -10.221] to (395.06, 312.72, -8.35) mm, rotated rx -180 ry 0 rz -179 deg; joints [6.688, -49.38, 82.17, 12.217, -33.39, -10.247]
  MoveL 372 to (395.06, 287.32, -8.35) mm, rotated rx -180 ry 0 rz -179 deg; joints [7.553, -49.203, 81.865, 13.803, -33.43, -11.587]
  MoveL 373 to (344.26, 287.32, -8.35) mm, rotated rx -180 ry 0 rz -179 deg; joints [7.758, -52.432, 87.37, 13.381, -35.681, -10.936]
  MoveL 374 to (344.26, 338.12, -8.35) mm, rotated rx -180 ry 0 rz -179 deg; joints [5.971, -52.757, 87.917, 10.295, -35.599, -8.401]
  MoveL 375 to (395.06, 338.12, -8.35) mm, rotated rx -180 ry 0 rz -179 deg; joints [5.82, -49.532, 82.431, 10.629, -33.353, -8.909]
  MoveL 376 to (395.06, 312.72, -8.35) mm, rotated rx -180 ry 0 rz -179 deg; joints [6.688, -49.38, 82.17, 12.217, -33.39, -10.247]
  MoveC 377 to (394.87, 312.27, -8.35) mm, rotated rx -180 ry 0 rz -179 deg; joints [6.704, -49.389, 82.186, 12.243, -33.4, -10.269] to (394.42, 312.09, -8.35) mm, rotated rx 180 ry 0 rz -179 deg; joints [6.712, -49.417, 82.234, 12.251, -33.421, -10.273]
  MoveL 378 to (393.79, 312.09, -8.35) mm, rotated rx 180 ry 0 rz -179 deg; joints [6.714, -49.458, 82.305, 12.245, -33.45, -10.264]
  MoveC 379 to (393.34, 312.09, -8.16) mm, rotated rx -180 ry 0 rz -179 deg; joints [6.715, -49.493, 82.35, 12.245, -33.461, -10.262] to (393.15, 312.08, -7.72) mm, rotated rx -180 ry 0 rz -179 deg; joints [6.716, -49.517, 82.358, 12.251, -33.446, -10.27]
  Set speed (500.0 mm/s)
  MoveL 380 to (393.15, 312.09, 6) mm, rotated rx 180 ry 0 rz -179 deg; joints [6.716, -49.888, 81.973, 12.5, -32.707, -10.567]
  MoveL 381 to (266.15, 313.36, 6) mm, rotated rx 180 ry 0 rz -179 deg; joints [7.139, -57.797, 95.123, 11.671, -37.904, -9.257]
  Set speed (25.4 mm/s)
  MoveL 382 to (266.15, 313.36, -3.54) mm, rotated rx -180 ry 0 rz -179 deg; joints [7.139, -57.499, 95.38, 11.529, -38.449, -9.076]
  MoveC 383 to (266.34, 313.36, -3.99) mm, rotated rx -180 ry 0 rz -179 deg; joints [7.138, -57.473, 95.374, 11.523, -38.468, -9.069] to (266.79, 313.36, -4.17) mm, rotated rx -180 ry 0 rz -179 deg; joints [7.136, -57.441, 95.336, 11.521, -38.462, -9.068]
  Set speed (50.8 mm/s)
  MoveL 384 to (267.42, 313.36, -4.17) mm, rotated rx -180 ry 0 rz -179 deg; joints [7.134, -57.403, 95.275, 11.523, -38.438, -9.073]
  MoveC 385 to (267.87, 313.17, -4.17) mm, rotated rx 180 ry 0 rz -179 deg; joints [7.139, -57.375, 95.23, 11.535, -38.422, -9.085] to (268.06, 312.72, -4.17) mm, rotated rx -180 ry 0 rz -179 deg; joints [7.155, -57.361, 95.207, 11.563, -38.416, -9.107]
  MoveL 386 to (268.06, 287.32, -4.18) mm, rotated rx -180 ry 0 rz -179 deg; joints [8.09, -57.186, 94.922, 13.074, -38.467, -10.306]
  MoveL 387 to (217.26, 287.32, -4.17) mm, rotated rx -180 ry 0 rz -179 deg; joints [8.329, -60.172, 99.713, 12.951, -40.268, -9.953]
  MoveL 388 to (217.26, 338.12, -4.17) mm, rotated rx -180 ry 0 rz -179 deg; joints [6.394, -60.502, 100.235, 9.944, -40.16, -7.631]
  MoveL 389 to (268.06, 338.12, -4.17) mm, rotated rx -180 ry 0 rz -179 deg; joints [6.217, -57.512, 95.451, 10.047, -38.369, -7.908]
  MoveL 390 to (268.06, 312.72, -4.17) mm, rotated rx -180 ry 0 rz -179 deg; joints [7.155, -57.361, 95.207, 11.563, -38.416, -9.107]
  MoveC 391 to (267.87, 312.27, -4.17) mm, rotated rx -180 ry 0 rz -179 deg; joints [7.172, -57.369, 95.22, 11.589, -38.424, -9.127] to (267.42, 312.09, -4.17) mm, rotated rx 180 ry 0 rz -179 deg; joints [7.181, -57.395, 95.262, 11.599, -38.441, -9.133]
  MoveL 392 to (266.79, 312.09, -4.17) mm, rotated rx 180 ry 0 rz -179 deg; joints [7.183, -57.433, 95.323, 11.597, -38.464, -9.128]
  MoveC 393 to (266.34, 312.09, -3.99) mm, rotated rx -180 ry 0 rz -179 deg; joints [7.185, -57.465, 95.361, 11.598, -38.47, -9.129] to (266.15, 312.08, -3.54) mm, rotated rx -180 ry 0 rz -179 deg; joints [7.186, -57.491, 95.367, 11.604, -38.451, -9.136]
  Set speed (500.0 mm/s)
  MoveL 394 to (266.15, 312.09, 5) mm, rotated rx -180 ry 0 rz -179 deg; joints [7.186, -57.758, 95.137, 11.732, -37.964, -9.299]
  MoveL 395 to (266.15, 313.36, 5) mm, rotated rx 180 ry 0 rz -179 deg; joints [7.139, -57.766, 95.15, 11.656, -37.961, -9.238]
  Set speed (25.4 mm/s)
  MoveL 396 to (266.15, 313.36, 1.83) mm, rotated rx -180 ry 0 rz -179 deg; joints [7.139, -57.667, 95.236, 11.608, -38.143, -9.177]
  MoveL 397 to (266.15, 313.36, -7.72) mm, rotated rx -180 ry 0 rz -179 deg; joints [7.139, -57.366, 95.491, 11.468, -38.687, -8.998]
  MoveC 398 to (266.34, 313.36, -8.16) mm, rotated rx 180 ry 0 rz -179 deg; joints [7.138, -57.341, 95.485, 11.462, -38.706, -8.991] to (266.79, 313.36, -8.35) mm, rotated rx -180 ry 0 rz -179 deg; joints [7.136, -57.308, 95.446, 11.461, -38.7, -8.991]
  Set speed (50.8 mm/s)
  MoveL 399 to (267.42, 313.36, -8.35) mm, rotated rx 180 ry 0 rz -179 deg; joints [7.134, -57.271, 95.385, 11.462, -38.676, -8.995]
  MoveC 400 to (267.87, 313.17, -8.35) mm, rotated rx -180 ry 0 rz -179 deg; joints [7.139, -57.243, 95.34, 11.475, -38.66, -9.007] to (268.06, 312.72, -8.35) mm, rotated rx -180 ry 0 rz -179 deg; joints [7.155, -57.229, 95.317, 11.502, -38.654, -9.029]
  MoveL 401 to (268.06, 287.32, -8.35) mm, rotated rx 180 ry 0 rz -179 deg; joints [8.09, -57.054, 95.033, 13.006, -38.703, -10.218]
  MoveL 402 to (217.26, 287.32, -8.35) mm, rotated rx 180 ry 0 rz -179 deg; joints [8.329, -60.033, 99.823, 12.886, -40.51, -9.867]
  MoveL 403 to (217.26, 338.12, -8.35) mm, rotated rx -180 ry 0 rz -179 deg; joints [6.394, -60.362, 100.345, 9.893, -40.406, -7.565]
  MoveL 404 to (268.06, 338.12, -8.35) mm, rotated rx -180 ry 0 rz -179 deg; joints [6.217, -57.379, 95.561, 9.994, -38.609, -7.84]
  MoveL 405 to (268.06, 312.72, -8.35) mm, rotated rx -180 ry 0 rz -179 deg; joints [7.155, -57.229, 95.317, 11.502, -38.654, -9.029]
  MoveC 406 to (267.87, 312.27, -8.35) mm, rotated rx -180 ry 0 rz -179 deg; joints [7.172, -57.237, 95.331, 11.528, -38.662, -9.049] to (267.42, 312.08, -8.35) mm, rotated rx -180 ry 0 rz -179 deg; joints [7.181, -57.263, 95.372, 11.538, -38.679, -9.055]
  MoveL 407 to (266.79, 312.09, -8.35) mm, rotated rx -180 ry 0 rz -179 deg; joints [7.183, -57.3, 95.433, 11.536, -38.702, -9.05]
  MoveC 408 to (266.34, 312.09, -8.16) mm, rotated rx 180 ry 0 rz -179 deg; joints [7.185, -57.333, 95.472, 11.537, -38.708, -9.051] to (266.15, 312.09, -7.72) mm, rotated rx -180 ry 0 rz -179 deg; joints [7.186, -57.358, 95.478, 11.543, -38.689, -9.058]
  Set speed (500.0 mm/s)
  MoveL 409 to (266.15, 312.09, 6) mm, rotated rx -180 ry 0 rz -179 deg; joints [7.186, -57.789, 95.109, 11.747, -37.907, -9.318]
  MoveL 410 to (139.15, 313.36, 6) mm, rotated rx 180 ry 0 rz -179 deg; joints [7.688, -65.217, 106.686, 11.522, -42.049, -8.608]
  Set speed (25.4 mm/s)
  MoveL 411 to (139.15, 313.36, -3.54) mm, rotated rx 180 ry 0 rz -179 deg; joints [7.688, -64.877, 106.945, 11.391, -42.636, -8.431]
  MoveC 412 to (139.34, 313.36, -3.99) mm, rotated rx -180 ry 0 rz -179 deg; joints [7.687, -64.85, 106.941, 11.385, -42.658, -8.423] to (139.79, 313.36, -4.17) mm, rotated rx 180 ry 0 rz -179 deg; joints [7.685, -64.817, 106.907, 11.382, -42.656, -8.422]
  Set speed (50.8 mm/s)
  MoveL 413 to (140.42, 313.36, -4.18) mm, rotated rx -180 ry 0 rz -179 deg; joints [7.682, -64.781, 106.852, 11.382, -42.638, -8.424]
  MoveC 414 to (140.87, 313.17, -4.18) mm, rotated rx -180 ry 0 rz -179 deg; joints [7.687, -64.754, 106.812, 11.393, -42.625, -8.434] to (141.06, 312.72, -4.17) mm, rotated rx 180 ry 0 rz -179 deg; joints [7.705, -64.741, 106.791, 11.419, -42.621, -8.454]
  MoveL 415 to (141.06, 287.32, -4.17) mm, rotated rx 180 ry 0 rz -179 deg; joints [8.721, -64.557, 106.513, 12.923, -42.687, -9.573]
  MoveL 416 to (90.26, 287.32, -4.17) mm, rotated rx 180 ry 0 rz -179 deg; joints [9.006, -67.446, 110.827, 12.994, -44.123, -9.406]
  MoveL 417 to (90.26, 338.12, -4.17) mm, rotated rx -180 ry 0 rz -179 deg; joints [6.895, -67.799, 111.343, 9.956, -43.979, -7.199]
  MoveL 418 to (141.06, 338.12, -4.17) mm, rotated rx -180 ry 0 rz -179 deg; joints [6.684, -64.898, 107.029, 9.909, -42.56, -7.332]
  MoveL 419 to (141.06, 312.72, -4.17) mm, rotated rx 180 ry 0 rz -179 deg; joints [7.705, -64.741, 106.791, 11.419, -42.621, -8.454]
  MoveC 420 to (140.87, 312.27, -4.17) mm, rotated rx 180 ry 0 rz -179 deg; joints [7.723, -64.748, 106.802, 11.446, -42.627, -8.473] to (140.42, 312.09, -4.17) mm, rotated rx -180 ry 0 rz -179 deg; joints [7.733, -64.773, 106.839, 11.457, -42.641, -8.48]
  MoveL 421 to (139.79, 312.09, -4.18) mm, rotated rx -180 ry 0 rz -179 deg; joints [7.736, -64.809, 106.894, 11.458, -42.66, -8.478]
  MoveC 422 to (139.34, 312.09, -3.99) mm, rotated rx -180 ry 0 rz -179 deg; joints [7.738, -64.841, 106.928, 11.461, -42.661, -8.48] to (139.15, 312.09, -3.54) mm, rotated rx 180 ry 0 rz -179 deg; joints [7.739, -64.868, 106.932, 11.467, -42.639, -8.487]
  Set speed (500.0 mm/s)
  MoveL 423 to (139.15, 312.09, 5) mm, rotated rx 180 ry 0 rz -179 deg; joints [7.739, -65.173, 106.701, 11.584, -42.114, -8.646]
  MoveL 424 to (139.15, 313.36, 5) mm, rotated rx -180 ry 0 rz -179 deg; joints [7.688, -65.182, 106.714, 11.508, -42.11, -8.589]
  Set speed (25.4 mm/s)
  MoveL 425 to (139.15, 313.36, 1.82) mm, rotated rx 180 ry 0 rz -179 deg; joints [7.688, -65.069, 106.801, 11.464, -42.306, -8.53]
  MoveL 426 to (139.15, 313.36, -7.72) mm, rotated rx 180 ry 0 rz -179 deg; joints [7.688, -64.726, 107.056, 11.336, -42.893, -8.355]
  MoveC 427 to (139.34, 313.36, -8.16) mm, rotated rx -180 ry 0 rz -179 deg; joints [7.687, -64.699, 107.052, 11.329, -42.915, -8.348] to (139.79, 313.36, -8.35) mm, rotated rx 180 ry 0 rz -179 deg; joints [7.685, -64.666, 107.018, 11.327, -42.913, -8.346]
  Set speed (50.8 mm/s)
  MoveL 428 to (140.42, 313.36, -8.35) mm, rotated rx 180 ry 0 rz -179 deg; joints [7.682, -64.63, 106.963, 11.326, -42.894, -8.348]
  MoveC 429 to (140.87, 313.17, -8.35) mm, rotated rx -180 ry 0 rz -179 deg; joints [7.687, -64.603, 106.922, 11.337, -42.881, -8.358] to (141.06, 312.72, -8.35) mm, rotated rx -180 ry 0 rz -179 deg; joints [7.705, -64.59, 106.902, 11.363, -42.877, -8.378]
  MoveL 430 to (141.06, 287.32, -8.35) mm, rotated rx -180 ry 0 rz -179 deg; joints [8.721, -64.407, 106.623, 12.86, -42.942, -9.488]
  MoveL 431 to (90.26, 287.32, -8.35) mm, rotated rx 180 ry 0 rz -179 deg; joints [9.006, -67.288, 110.939, 12.932, -44.386, -9.319]
  MoveL 432 to (90.26, 338.12, -8.35) mm, rotated rx 180 ry 0 rz -179 deg; joints [6.895, -67.64, 111.455, 9.907, -44.246, -7.132]
  MoveL 433 to (141.06, 338.12, -8.35) mm, rotated rx -180 ry 0 rz -179 deg; joints [6.684, -64.747, 107.14, 9.86, -42.818, -7.266]
  MoveL 434 to (141.06, 312.72, -8.35) mm, rotated rx -180 ry 0 rz -179 deg; joints [7.705, -64.59, 106.902, 11.363, -42.877, -8.378]
  MoveC 435 to (140.87, 312.27, -8.35) mm, rotated rx -180 ry 0 rz -179 deg; joints [7.723, -64.597, 106.913, 11.39, -42.884, -8.397] to (140.42, 312.09, -8.35) mm, rotated rx -180 ry 0 rz -179 deg; joints [7.733, -64.622, 106.95, 11.401, -42.897, -8.404]
  MoveL 436 to (139.79, 312.09, -8.35) mm, rotated rx 180 ry 0 rz -179 deg; joints [7.736, -64.658, 107.005, 11.402, -42.916, -8.401]
  MoveC 437 to (139.34, 312.09, -8.16) mm, rotated rx -180 ry 0 rz -179 deg; joints [7.738, -64.69, 107.039, 11.404, -42.918, -8.403] to (139.15, 312.09, -7.72) mm, rotated rx -180 ry 0 rz -179 deg; joints [7.739, -64.717, 107.043, 11.411, -42.896, -8.411]
  Set speed (500.0 mm/s)
  MoveL 438 to (139.15, 312.09, 6) mm, rotated rx 180 ry 0 rz -179 deg; joints [7.739, -65.209, 106.674, 11.598, -42.052, -8.665]
  MoveL 439 to (139.15, 131.49, 6) mm, rotated rx -180 ry 0 rz -179 deg; joints [14.848, -63.332, 103.827, 22.208, -42.687, -16.704]
  Set speed (25.4 mm/s)
  MoveL 440 to (139.15, 131.49, -3.54) mm, rotated rx -180 ry 0 rz -179 deg; joints [14.848, -63.002, 104.084, 21.97, -43.231, -16.38]
  MoveC 441 to (139.34, 131.49, -3.99) mm, rotated rx 180 ry 0 rz -179 deg; joints [14.846, -62.976, 104.08, 21.959, -43.251, -16.366] to (139.79, 131.49, -4.17) mm, rotated rx 180 ry 0 rz -179 deg; joints [14.842, -62.944, 104.046, 21.954, -43.247, -16.363]
  Set speed (50.8 mm/s)
  MoveL 442 to (140.42, 131.49, -4.18) mm, rotated rx -180 ry 0 rz -179 deg; joints [14.836, -62.908, 103.991, 21.954, -43.228, -16.368]
  MoveC 443 to (140.87, 131.3, -4.17) mm, rotated rx -180 ry 0 rz -179 deg; joints [14.839, -62.881, 103.948, 21.964, -43.215, -16.379] to (141.06, 130.85, -4.17) mm, rotated rx -180 ry 0 rz -179 deg; joints [14.854, -62.864, 103.922, 21.989, -43.211, -16.4]
  MoveL 444 to (141.06, 105.45, -4.17) mm, rotated rx -180 ry 0 rz -179 deg; joints [15.824, -62.5, 103.359, 23.424, -43.31, -17.497]
  MoveL 445 to (90.26, 105.45, -4.17) mm, rotated rx -180 ry 0 rz -179 deg; joints [16.353, -65.33, 107.68, 23.536, -44.834, -17.165]
  MoveL 446 to (90.26, 156.25, -4.18) mm, rotated rx 180 ry 0 rz -179 deg; joints [14.341, -66.053, 108.763, 20.653, -44.611, -15.02]
  MoveL 447 to (141.06, 156.25, -4.17) mm, rotated rx -180 ry 0 rz -179 deg; joints [13.877, -63.204, 104.446, 20.543, -43.115, -15.299]
  MoveL 448 to (141.06, 130.85, -4.17) mm, rotated rx -180 ry 0 rz -179 deg; joints [14.854, -62.864, 103.922, 21.989, -43.211, -16.4]
  MoveC 449 to (140.87, 130.4, -4.18) mm, rotated rx 180 ry 0 rz -179 deg; joints [14.873, -62.868, 103.929, 22.015, -43.218, -16.418] to (140.42, 130.22, -4.17) mm, rotated rx -180 ry 0 rz -179 deg; joints [14.885, -62.891, 103.964, 22.026, -43.233, -16.423]
  MoveL 450 to (139.79, 130.22, -4.18) mm, rotated rx -180 ry 0 rz -179 deg; joints [14.891, -62.927, 104.019, 22.026, -43.252, -16.418]
  MoveC 451 to (139.34, 130.22, -3.99) mm, rotated rx 180 ry 0 rz -179 deg; joints [14.895, -62.958, 104.053, 22.031, -43.256, -16.421] to (139.15, 130.22, -3.54) mm, rotated rx -180 ry 0 rz -179 deg; joints [14.897, -62.984, 104.057, 22.043, -43.236, -16.435]
  Set speed (500.0 mm/s)
  MoveL 452 to (139.15, 130.22, 5) mm, rotated rx 180 ry 0 rz -179 deg; joints [14.897, -63.28, 103.827, 22.255, -42.749, -16.725]
  MoveL 453 to (139.15, 131.49, 5) mm, rotated rx -180 ry 0 rz -179 deg; joints [14.848, -63.297, 103.854, 22.182, -42.744, -16.67]
  Set speed (25.4 mm/s)
  MoveL 454 to (139.15, 131.49, 1.83) mm, rotated rx -180 ry 0 rz -179 deg; joints [14.848, -63.188, 103.94, 22.103, -42.925, -16.561]
  MoveL 455 to (139.15, 131.49, -7.71) mm, rotated rx -180 ry 0 rz -179 deg; joints [14.848, -62.856, 104.194, 21.869, -43.469, -16.241]
  MoveC 456 to (139.34, 131.49, -8.16) mm, rotated rx 180 ry 0 rz -179 deg; joints [14.846, -62.83, 104.19, 21.858, -43.489, -16.227] to (139.79, 131.49, -8.35) mm, rotated rx 180 ry 0 rz -179 deg; joints [14.842, -62.798, 104.156, 21.853, -43.485, -16.224]
  Set speed (50.8 mm/s)
  MoveL 457 to (140.42, 131.49, -8.35) mm, rotated rx 180 ry 0 rz -179 deg; joints [14.836, -62.762, 104.101, 21.852, -43.466, -16.228]
  MoveC 458 to (140.87, 131.3, -8.35) mm, rotated rx -180 ry 0 rz -179 deg; joints [14.839, -62.735, 104.058, 21.862, -43.452, -16.239] to (141.06, 130.85, -8.35) mm, rotated rx -180 ry 0 rz -179 deg; joints [14.854, -62.718, 104.032, 21.887, -43.448, -16.26]
  MoveL 459 to (141.06, 105.45, -8.35) mm, rotated rx -180 ry 0 rz -179 deg; joints [15.824, -62.355, 103.469, 23.317, -43.544, -17.35]
  MoveL 460 to (90.26, 105.45, -8.35) mm, rotated rx 180 ry 0 rz -179 deg; joints [16.353, -65.177, 107.79, 23.431, -45.076, -17.016]
  MoveL 461 to (90.26, 156.25, -8.35) mm, rotated rx -180 ry 0 rz -179 deg; joints [14.341, -65.898, 108.874, 20.558, -44.859, -14.888]
  MoveL 462 to (141.06, 156.25, -8.35) mm, rotated rx -180 ry 0 rz -179 deg; joints [13.877, -63.057, 104.556, 20.447, -43.356, -15.168]
  MoveL 463 to (141.06, 130.85, -8.35) mm, rotated rx -180 ry 0 rz -179 deg; joints [14.854, -62.718, 104.032, 21.887, -43.448, -16.26]
  MoveC 464 to (140.87, 130.4, -8.35) mm, rotated rx -180 ry 0 rz -179 deg; joints [14.873, -62.722, 104.039, 21.913, -43.456, -16.278] to (140.42, 130.22, -8.35) mm, rotated rx 180 ry 0 rz -179 deg; joints [14.885, -62.745, 104.074, 21.924, -43.47, -16.283]
  MoveL 465 to (139.79, 130.21, -8.35) mm, rotated rx -180 ry 0 rz -179 deg; joints [14.891, -62.78, 104.129, 21.925, -43.49, -16.278]
  MoveC 466 to (139.34, 130.22, -8.16) mm, rotated rx 180 ry 0 rz -179 deg; joints [14.895, -62.812, 104.163, 21.93, -43.493, -16.281] to (139.15, 130.22, -7.72) mm, rotated rx -180 ry 0 rz -179 deg; joints [14.897, -62.838, 104.167, 21.941, -43.474, -16.295]
  Set speed (500.0 mm/s)
  MoveL 467 to (139.15, 130.22, 6) mm, rotated rx -180 ry 0 rz -179 deg; joints [14.897, -63.314, 103.799, 22.28, -42.692, -16.76]
  MoveL 468 to (266.15, 131.49, 6) mm, rotated rx 180 ry 0 rz -179 deg; joints [13.741, -55.987, 92.183, 22.493, -38.38, -17.983]
  Set speed (25.4 mm/s)
  MoveL 469 to (266.15, 131.49, -3.54) mm, rotated rx -180 ry 0 rz -179 deg; joints [13.741, -55.698, 92.442, 22.232, -38.887, -17.649]
  MoveC 470 to (266.34, 131.49, -3.99) mm, rotated rx 180 ry 0 rz -179 deg; joints [13.739, -55.674, 92.436, 22.221, -38.904, -17.636] to (266.79, 131.49, -4.17) mm, rotated rx 180 ry 0 rz -179 deg; joints [13.736, -55.641, 92.397, 22.219, -38.896, -17.636]
  Set speed (50.8 mm/s)
  MoveL 471 to (267.42, 131.48, -4.17) mm, rotated rx -180 ry 0 rz -179 deg; joints [13.73, -55.604, 92.335, 22.222, -38.872, -17.644]
  MoveC 472 to (267.87, 131.3, -4.17) mm, rotated rx 180 ry 0 rz -179 deg; joints [13.733, -55.575, 92.287, 22.236, -38.856, -17.659] to (268.06, 130.85, -4.18) mm, rotated rx -180 ry 0 rz -179 deg; joints [13.748, -55.558, 92.259, 22.263, -38.85, -17.683]
  MoveL 473 to (268.06, 105.45, -4.18) mm, rotated rx -180 ry 0 rz -179 deg; joints [14.646, -55.205, 91.677, 23.732, -38.921, -18.883]
  MoveL 474 to (217.26, 105.45, -4.17) mm, rotated rx -180 ry 0 rz -179 deg; joints [15.094, -58.173, 96.519, 23.496, -40.781, -18.221]
  MoveL 475 to (217.26, 156.25, -4.18) mm, rotated rx -180 ry 0 rz -179 deg; joints [13.236, -58.859, 97.622, 20.591, -40.621, -15.916]
  MoveL 476 to (268.06, 156.25, -4.18) mm, rotated rx -180 ry 0 rz -179 deg; joints [12.843, -55.886, 92.799, 20.787, -38.781, -16.485]
  MoveL 477 to (268.06, 130.85, -4.18) mm, rotated rx -180 ry 0 rz -179 deg; joints [13.748, -55.558, 92.259, 22.263, -38.85, -17.683]
  MoveC 478 to (267.87, 130.4, -4.18) mm, rotated rx 180 ry 0 rz -179 deg; joints [13.765, -55.563, 92.267, 22.288, -38.858, -17.702] to (267.42, 130.21, -4.18) mm, rotated rx 180 ry 0 rz -179 deg; joints [13.776, -55.587, 92.307, 22.296, -38.876, -17.704]
  MoveL 479 to (266.79, 130.22, -4.18) mm, rotated rx -180 ry 0 rz -179 deg; joints [13.781, -55.624, 92.369, 22.292, -38.9, -17.696]
  MoveC 480 to (266.34, 130.22, -3.99) mm, rotated rx 180 ry 0 rz -179 deg; joints [13.784, -55.657, 92.408, 22.295, -38.907, -17.696] to (266.15, 130.21, -3.54) mm, rotated rx -180 ry 0 rz -179 deg; joints [13.786, -55.681, 92.414, 22.306, -38.89, -17.709]
  Set speed (500.0 mm/s)
  MoveL 481 to (266.15, 130.21, 5) mm, rotated rx -180 ry 0 rz -179 deg; joints [13.786, -55.94, 92.182, 22.54, -38.437, -18.009]
  MoveL 482 to (266.15, 131.49, 5) mm, rotated rx -180 ry 0 rz -179 deg; joints [13.741, -55.957, 92.21, 22.465, -38.433, -17.948]
  Set speed (25.4 mm/s)
  MoveL 483 to (266.15, 131.49, 1.83) mm, rotated rx -180 ry 0 rz -179 deg; joints [13.741, -55.862, 92.297, 22.378, -38.602, -17.836]
  MoveL 484 to (266.15, 131.49, -7.71) mm, rotated rx -180 ry 0 rz -179 deg; joints [13.741, -55.57, 92.553, 22.121, -39.108, -17.506]
  MoveC 485 to (266.34, 131.49, -8.16) mm, rotated rx 180 ry 0 rz -179 deg; joints [13.739, -55.545, 92.547, 22.11, -39.125, -17.493] to (266.79, 131.49, -8.35) mm, rotated rx 180 ry 0 rz -179 deg; joints [13.736, -55.513, 92.508, 22.107, -39.118, -17.493]
  Set speed (50.8 mm/s)
  MoveL 486 to (267.42, 131.49, -8.35) mm, rotated rx -180 ry 0 rz -179 deg; joints [13.73, -55.476, 92.446, 22.111, -39.094, -17.501]
  MoveC 487 to (267.87, 131.3, -8.35) mm, rotated rx 180 ry 0 rz -179 deg; joints [13.733, -55.447, 92.398, 22.124, -39.077, -17.516] to (268.06, 130.85, -8.35) mm, rotated rx -180 ry 0 rz -179 deg; joints [13.748, -55.43, 92.37, 22.151, -39.071, -17.539]
  MoveL 488 to (268.06, 105.45, -8.35) mm, rotated rx 180 ry 0 rz -179 deg; joints [14.646, -55.077, 91.788, 23.614, -39.139, -18.731]
  MoveL 489 to (217.26, 105.45, -8.35) mm, rotated rx 180 ry 0 rz -179 deg; joints [15.094, -58.038, 96.629, 23.384, -41.005, -18.072]
  MoveL 490 to (217.26, 156.25, -8.35) mm, rotated rx 180 ry 0 rz -179 deg; joints [13.236, -58.723, 97.732, 20.491, -40.852, -15.784]
  MoveL 491 to (268.06, 156.25, -8.35) mm, rotated rx -180 ry 0 rz -179 deg; joints [12.843, -55.757, 92.91, 20.682, -39.005, -16.349]
  MoveL 492 to (268.06, 130.85, -8.35) mm, rotated rx -180 ry 0 rz -179 deg; joints [13.748, -55.43, 92.37, 22.151, -39.071, -17.539]
  MoveC 493 to (267.87, 130.4, -8.35) mm, rotated rx 180 ry 0 rz -179 deg; joints [13.765, -55.435, 92.378, 22.176, -39.08, -17.558] to (267.42, 130.21, -8.35) mm, rotated rx -180 ry 0 rz -179 deg; joints [13.776, -55.459, 92.418, 22.184, -39.097, -17.561]
  MoveL 494 to (266.79, 130.22, -8.35) mm, rotated rx 180 ry 0 rz -179 deg; joints [13.781, -55.496, 92.48, 22.181, -39.121, -17.552]
  MoveC 495 to (266.34, 130.21, -8.16) mm, rotated rx -180 ry 0 rz -179 deg; joints [13.784, -55.528, 92.519, 22.183, -39.128, -17.552] to (266.15, 130.22, -7.72) mm, rotated rx 180 ry 0 rz -179 deg; joints [13.786, -55.553, 92.525, 22.194, -39.112, -17.565]
  Set speed (500.0 mm/s)
  MoveL 496 to (266.15, 130.22, 6) mm, rotated rx 180 ry 0 rz -179 deg; joints [13.786, -55.97, 92.155, 22.567, -38.384, -18.044]
  MoveL 497 to (393.15, 131.48, 6) mm, rotated rx -180 ry 0 rz -179 deg; joints [12.795, -48.053, 78.818, 23.94, -33.077, -20.406]
  Set speed (25.4 mm/s)
  MoveL 498 to (393.15, 131.48, -3.54) mm, rotated rx -180 ry 0 rz -179 deg; joints [12.795, -47.806, 79.093, 23.62, -33.555, -20.023]
  MoveC 499 to (393.34, 131.49, -3.99) mm, rotated rx 180 ry 0 rz -179 deg; joints [12.794, -47.782, 79.085, 23.608, -33.569, -20.01] to (393.79, 131.49, -4.17) mm, rotated rx 180 ry 0 rz -179 deg; joints [12.791, -47.748, 79.039, 23.61, -33.557, -20.014]
  Set speed (50.8 mm/s)
  MoveL 500 to (394.42, 131.49, -4.18) mm, rotated rx 180 ry 0 rz -179 deg; joints [12.786, -47.706, 78.966, 23.621, -33.527, -20.03]
  MoveC 501 to (394.87, 131.3, -4.17) mm, rotated rx -180 ry 0 rz -179 deg; joints [12.789, -47.674, 78.91, 23.641, -33.507, -20.052] to (395.06, 130.85, -4.17) mm, rotated rx -180 ry 0 rz -179 deg; joints [12.803, -47.655, 78.878, 23.672, -33.499, -20.081]
  MoveL 502 to (395.06, 105.45, -4.17) mm, rotated rx -180 ry 0 rz -179 deg; joints [13.639, -47.292, 78.246, 25.255, -33.551, -21.462]
  MoveL 503 to (344.26, 105.45, -4.17) mm, rotated rx -180 ry 0 rz -179 deg; joints [14.023, -50.563, 83.885, 24.449, -35.836, -20.233]
  MoveL 504 to (344.26, 156.25, -4.17) mm, rotated rx -180 ry 0 rz -179 deg; joints [12.298, -51.25, 85.054, 21.398, -35.72, -17.648]
  MoveL 505 to (395.06, 156.25, -4.18) mm, rotated rx -180 ry 0 rz -179 deg; joints [11.962, -47.992, 79.463, 22.088, -33.448, -18.706]
  MoveL 506 to (395.06, 130.85, -4.17) mm, rotated rx -180 ry 0 rz -179 deg; joints [12.803, -47.655, 78.878, 23.672, -33.499, -20.081]
  MoveC 507 to (394.87, 130.4, -4.18) mm, rotated rx 180 ry 0 rz -179 deg; joints [12.819, -47.661, 78.889, 23.697, -33.508, -20.1] to (394.42, 130.21, -4.17) mm, rotated rx -180 ry 0 rz -179 deg; joints [12.828, -47.688, 78.936, 23.7, -33.53, -20.099]
  MoveL 508 to (393.79, 130.22, -4.17) mm, rotated rx 180 ry 0 rz -179 deg; joints [12.832, -47.73, 79.008, 23.689, -33.56, -20.083]
  MoveC 509 to (393.34, 130.22, -3.99) mm, rotated rx -180 ry 0 rz -179 deg; joints [12.836, -47.765, 79.055, 23.687, -33.571, -20.079] to (393.15, 130.22, -3.54) mm, rotated rx 180 ry 0 rz -179 deg; joints [12.837, -47.789, 79.063, 23.699, -33.558, -20.092]
  Set speed (500.0 mm/s)
  MoveL 510 to (393.15, 130.21, 5) mm, rotated rx 180 ry 0 rz -179 deg; joints [12.837, -48.01, 78.817, 23.986, -33.13, -20.435]
  MoveL 511 to (393.15, 131.48, 5) mm, rotated rx -180 ry 0 rz -179 deg; joints [12.795, -48.028, 78.847, 23.906, -33.127, -20.366]
  Set speed (25.4 mm/s)
  MoveL 512 to (393.15, 131.48, 1.83) mm, rotated rx -180 ry 0 rz -179 deg; joints [12.795, -47.946, 78.94, 23.798, -33.287, -20.237]
  MoveL 513 to (393.15, 131.48, -7.72) mm, rotated rx -180 ry 0 rz -179 deg; joints [12.795, -47.697, 79.211, 23.483, -33.764, -19.859]
  MoveC 514 to (393.34, 131.49, -8.16) mm, rotated rx -180 ry 0 rz -179 deg; joints [12.794, -47.672, 79.203, 23.472, -33.777, -19.846] to (393.79, 131.49, -8.35) mm, rotated rx 180 ry 0 rz -179 deg; joints [12.791, -47.638, 79.156, 23.473, -33.766, -19.85]
  Set speed (50.8 mm/s)
  MoveL 515 to (394.42, 131.49, -8.35) mm, rotated rx -180 ry 0 rz -179 deg; joints [12.786, -47.596, 79.084, 23.484, -33.736, -19.866]
  MoveC 516 to (394.87, 131.3, -8.35) mm, rotated rx -180 ry 0 rz -179 deg; joints [12.789, -47.564, 79.028, 23.504, -33.715, -19.887] to (395.06, 130.85, -8.35) mm, rotated rx 180 ry 0 rz -179 deg; joints [12.803, -47.546, 78.996, 23.535, -33.707, -19.916]
  MoveL 517 to (395.06, 105.45, -8.35) mm, rotated rx -180 ry 0 rz -179 deg; joints [13.639, -47.183, 78.364, 25.11, -33.756, -21.288]
  MoveL 518 to (344.26, 105.45, -8.35) mm, rotated rx -180 ry 0 rz -179 deg; joints [14.023, -50.447, 83.999, 24.318, -36.046, -20.071]
  MoveL 519 to (344.26, 156.25, -8.35) mm, rotated rx 180 ry 0 rz -179 deg; joints [12.298, -51.132, 85.167, 21.281, -35.936, -17.504]
  MoveL 520 to (395.06, 156.25, -8.35) mm, rotated rx -180 ry 0 rz -179 deg; joints [11.962, -47.882, 79.58, 21.959, -33.659, -18.552]
  MoveL 521 to (395.06, 130.85, -8.35) mm, rotated rx 180 ry 0 rz -179 deg; joints [12.803, -47.546, 78.996, 23.535, -33.707, -19.916]
  MoveC 522 to (394.87, 130.4, -8.35) mm, rotated rx -180 ry 0 rz -179 deg; joints [12.819, -47.552, 79.007, 23.559, -33.717, -19.936] to (394.42, 130.22, -8.35) mm, rotated rx -180 ry 0 rz -179 deg; joints [12.828, -47.579, 79.054, 23.563, -33.738, -19.934]
  MoveL 523 to (393.79, 130.22, -8.35) mm, rotated rx -180 ry 0 rz -179 deg; joints [12.832, -47.621, 79.126, 23.552, -33.768, -19.918]
  MoveC 524 to (393.34, 130.22, -8.16) mm, rotated rx 180 ry 0 rz -179 deg; joints [12.836, -47.655, 79.172, 23.55, -33.78, -19.914] to (393.15, 130.22, -7.72) mm, rotated rx -180 ry 0 rz -179 deg; joints [12.837, -47.679, 79.181, 23.562, -33.766, -19.927]
  Set speed (500.0 mm/s)
  MoveL 525 to (393.15, 130.22, 6) mm, rotated rx 180 ry 0 rz -179 deg; joints [12.837, -48.036, 78.788, 24.02, -33.08, -20.476]
  MoveL 526 to (393.15, -54.85, 6) mm, rotated rx 180 ry 0 rz -179 deg; joints [18.796, -44.736, 73.023, 35.686, -33.528, -30.91]
  Set speed (25.4 mm/s)
  MoveL 527 to (393.15, -54.85, -3.54) mm, rotated rx -180 ry 0 rz -179 deg; joints [18.796, -44.507, 73.311, 35.237, -33.949, -30.37]
  MoveC 528 to (393.34, -54.85, -3.99) mm, rotated rx 180 ry 0 rz -179 deg; joints [18.794, -44.483, 73.302, 35.222, -33.96, -30.352] to (393.79, -54.85, -4.17) mm, rotated rx -180 ry 0 rz -179 deg; joints [18.79, -44.448, 73.253, 35.227, -33.946, -30.36]
  Set speed (50.8 mm/s)
  MoveL 529 to (394.42, -54.85, -4.17) mm, rotated rx 180 ry 0 rz -179 deg; joints [18.784, -44.405, 73.177, 35.245, -33.916, -30.387]
  MoveC 530 to (394.87, -55.04, -4.17) mm, rotated rx -180 ry 0 rz -179 deg; joints [18.785, -44.37, 73.116, 35.27, -33.895, -30.416] to (395.06, -55.49, -4.18) mm, rotated rx -180 ry 0 rz -179 deg; joints [18.797, -44.348, 73.076, 35.304, -33.887, -30.45]
  MoveL 531 to (395.06, -80.89, -4.18) mm, rotated rx -180 ry 0 rz -179 deg; joints [19.587, -43.776, 72.062, 36.902, -33.939, -31.921]
  MoveL 532 to (344.26, -80.89, -4.17) mm, rotated rx 180 ry 0 rz -179 deg; joints [20.131, -47.146, 77.993, 35.561, -36.283, -29.954]
  MoveL 533 to (344.26, -30.09, -4.17) mm, rotated rx -180 ry 0 rz -179 deg; joints [18.504, -48.222, 79.861, 32.537, -36.161, -27.252]
  MoveL 534 to (395.06, -30.09, -4.17) mm, rotated rx -180 ry 0 rz -179 deg; joints [18, -44.889, 74.032, 33.711, -33.834, -28.996]
  MoveL 535 to (395.06, -55.49, -4.18) mm, rotated rx -180 ry 0 rz -179 deg; joints [18.797, -44.348, 73.076, 35.304, -33.887, -30.45]
  MoveC 536 to (394.87, -55.94, -4.18) mm, rotated rx 180 ry 0 rz -179 deg; joints [18.813, -44.351, 73.081, 35.327, -33.897, -30.468] to (394.42, -56.12, -4.17) mm, rotated rx -180 ry 0 rz -179 deg; joints [18.823, -44.377, 73.128, 35.325, -33.918, -30.46]
  MoveL 537 to (393.79, -56.12, -4.17) mm, rotated rx -180 ry 0 rz -179 deg; joints [18.83, -44.42, 73.204, 35.306, -33.949, -30.433]
  MoveC 538 to (393.34, -56.12, -3.99) mm, rotated rx -180 ry 0 rz -179 deg; joints [18.834, -44.455, 73.253, 35.302, -33.962, -30.425] to (393.15, -56.12, -3.54) mm, rotated rx -180 ry 0 rz -179 deg; joints [18.836, -44.479, 73.262, 35.317, -33.951, -30.443]
  Set speed (500.0 mm/s)
  MoveL 539 to (393.15, -56.12, 5) mm, rotated rx -180 ry 0 rz -179 deg; joints [18.836, -44.684, 73.004, 35.719, -33.575, -30.926]
  MoveL 540 to (393.15, -54.85, 5) mm, rotated rx -180 ry 0 rz -179 deg; joints [18.796, -44.712, 73.054, 35.639, -33.572, -30.852]
  Set speed (25.4 mm/s)
  MoveL 541 to (393.15, -54.85, 1.83) mm, rotated rx -180 ry 0 rz -179 deg; joints [18.796, -44.636, 73.15, 35.488, -33.712, -30.671]
  MoveL 542 to (393.15, -54.85, -7.72) mm, rotated rx 180 ry 0 rz -179 deg; joints [18.796, -44.405, 73.434, 35.046, -34.133, -30.138]
  MoveC 543 to (393.34, -54.85, -8.16) mm, rotated rx -180 ry 0 rz -179 deg; joints [18.794, -44.381, 73.425, 35.03, -34.144, -30.121] to (393.79, -54.85, -8.35) mm, rotated rx -180 ry 0 rz -179 deg; joints [18.79, -44.346, 73.376, 35.035, -34.13, -30.129]
  Set speed (50.8 mm/s)
  MoveL 544 to (394.42, -54.85, -8.35) mm, rotated rx -180 ry 0 rz -179 deg; joints [18.784, -44.303, 73.3, 35.053, -34.1, -30.155]
  MoveC 545 to (394.87, -55.04, -8.35) mm, rotated rx 180 ry 0 rz -179 deg; joints [18.785, -44.268, 73.239, 35.078, -34.079, -30.184] to (395.06, -55.49, -8.35) mm, rotated rx -180 ry 0 rz -179 deg; joints [18.797, -44.246, 73.199, 35.112, -34.07, -30.218]
  MoveL 546 to (395.06, -80.89, -8.35) mm, rotated rx -180 ry 0 rz -179 deg; joints [19.587, -43.676, 72.187, 36.703, -34.119, -31.681]
  MoveL 547 to (344.26, -80.89, -8.35) mm, rotated rx -180 ry 0 rz -179 deg; joints [20.131, -47.038, 78.111, 35.382, -36.468, -29.732]
  MoveL 548 to (344.26, -30.09, -8.35) mm, rotated rx -180 ry 0 rz -179 deg; joints [18.504, -48.111, 79.978, 32.371, -36.354, -27.045]
  MoveL 549 to (395.06, -30.09, -8.35) mm, rotated rx -180 ry 0 rz -179 deg; joints [18, -44.786, 74.155, 33.526, -34.022, -28.772]
  MoveL 550 to (395.06, -55.49, -8.35) mm, rotated rx -180 ry 0 rz -179 deg; joints [18.797, -44.246, 73.199, 35.112, -34.07, -30.218]
  MoveC 551 to (394.87, -55.94, -8.35) mm, rotated rx -180 ry 0 rz -179 deg; joints [18.813, -44.249, 73.204, 35.134, -34.08, -30.236] to (394.42, -56.12, -8.35) mm, rotated rx -180 ry 0 rz -179 deg; joints [18.823, -44.275, 73.251, 35.133, -34.102, -30.228]
  MoveL 552 to (393.79, -56.12, -8.35) mm, rotated rx 180 ry 0 rz -179 deg; joints [18.83, -44.318, 73.327, 35.114, -34.133, -30.202]
  MoveC 553 to (393.34, -56.12, -8.16) mm, rotated rx -180 ry 0 rz -179 deg; joints [18.834, -44.353, 73.376, 35.11, -34.146, -30.194] to (393.15, -56.12, -7.72) mm, rotated rx -180 ry 0 rz -179 deg; joints [18.836, -44.377, 73.385, 35.125, -34.135, -30.211]
  Set speed (500.0 mm/s)
  MoveL 554 to (393.15, -56.12, 6) mm, rotated rx 180 ry 0 rz -179 deg; joints [18.836, -44.708, 72.974, 35.767, -33.531, -30.983]
  MoveL 555 to (266.15, -54.85, 6) mm, rotated rx 180 ry 0 rz -179 deg; joints [20.166, -52.803, 86.909, 33.223, -38.991, -26.979]
  Set speed (25.4 mm/s)
  MoveL 556 to (266.15, -54.85, -3.54) mm, rotated rx 180 ry 0 rz -179 deg; joints [20.166, -52.531, 87.172, 32.865, -39.44, -26.517]
  MoveC 557 to (266.34, -54.85, -3.99) mm, rotated rx 180 ry 0 rz -179 deg; joints [20.164, -52.507, 87.166, 32.851, -39.453, -26.5] to (266.79, -54.85, -4.17) mm, rotated rx 180 ry 0 rz -179 deg; joints [20.158, -52.475, 87.126, 32.849, -39.445, -26.501]
  Set speed (50.8 mm/s)
  MoveL 558 to (267.42, -54.85, -4.17) mm, rotated rx -180 ry 0 rz -179 deg; joints [20.151, -52.438, 87.063, 32.855, -39.42, -26.515]
  MoveC 559 to (267.87, -55.04, -4.18) mm, rotated rx -180 ry 0 rz -179 deg; joints [20.152, -52.407, 87.011, 32.87, -39.403, -26.534] to (268.06, -55.49, -4.17) mm, rotated rx 180 ry 0 rz -179 deg; joints [20.165, -52.387, 86.977, 32.898, -39.397, -26.56]
  MoveL 560 to (268.06, -80.89, -4.17) mm, rotated rx -180 ry 0 rz -179 deg; joints [21.006, -51.849, 86.069, 34.325, -39.473, -27.792]
  MoveL 561 to (217.26, -80.89, -4.17) mm, rotated rx -180 ry 0 rz -179 deg; joints [21.633, -54.814, 91.032, 33.871, -41.414, -26.72]
  MoveL 562 to (217.26, -30.09, -4.17) mm, rotated rx -180 ry 0 rz -179 deg; joints [19.898, -55.861, 92.758, 31.085, -41.238, -24.387]
  MoveL 563 to (268.06, -30.09, -4.17) mm, rotated rx -180 ry 0 rz -179 deg; joints [19.315, -52.899, 87.838, 31.466, -39.32, -25.335]
  MoveL 564 to (268.06, -55.49, -4.17) mm, rotated rx 180 ry 0 rz -179 deg; joints [20.165, -52.387, 86.977, 32.898, -39.397, -26.56]
